LIN {X 0,Y 235.118,Z 411.198,A -85,B 0,C 180,E1 -19815.606,E2 -19815.606} C_VEL
LIN {X 0,Y 235.013,Z 411.211,A -85,B 0,C 180,E1 -19819.205,E2 -19819.205} C_VEL
LIN {X 0,Y 234.964,Z 411.217,A -85,B 0,C 180,E1 -19822.882,E2 -19822.882} C_VEL
LIN {X 0,Y 234.971,Z 411.217,A -85,B 0,C 180,E1 -19826.657,E2 -19826.657} C_VEL
LIN {X 0,Y 234.956,Z 411.22,A -85,B 0,C 180,E1 -19831.565,E2 -19831.565} C_VEL
LIN {X 0,Y 234.996,Z 411.371,A -85,B 0,C 180,E1 -19832.57,E2 -19832.57} C_VEL
LIN {X 0,Y 235.541,Z 414.614,A -85,B 0,C 180,E1 -19836.638,E2 -19836.638} C_VEL
LIN {X 0,Y 236.198,Z 418.359,A -85,B 0,C 180,E1 -19840.89,E2 -19840.89} C_VEL
LIN {X 0,Y 237.06,Z 422.615,A -85,B 0,C 180,E1 -19845.359,E2 -19845.359} C_VEL
LIN {X 0,Y 237.901,Z 427.546,A -85,B 0,C 180,E1 -19850.116,E2 -19850.116} C_VEL
LIN {X 0,Y 237.366,Z 428.622,A -85,B 0,C 180,E1 -19851.017,E2 -19851.017} C_VEL
LIN {X 0,Y 234.575,Z 430.575,A -85,B 0,C 180,E1 -19852.411,E2 -19852.411} C_VEL
LIN {X 0,Y 231.461,Z 432.564,A -85,B 0,C 180,E1 -19853.829,E2 -19853.829} C_VEL
LIN {X 0,Y 230.488,Z 433.723,A -85,B 0,C 180,E1 -19854.763,E2 -19854.763} C_VEL
LIN {X 0,Y 229.679,Z 436.812,A -85,B 0,C 180,E1 -19857.317,E2 -19857.317} C_VEL
LIN {X 0,Y 233.039,Z 450.186,A -85,B 0,C 180,E1 -19858.643,E2 -19858.643} C_VEL
LIN {X 0,Y 235.255,Z 462.15,A -85,B 0,C 180,E1 -19860.037,E2 -19860.037} C_VEL
LIN {X 0,Y 236.595,Z 473.99,A -85,B 0,C 180,E1 -19861.622,E2 -19861.622} C_VEL
LIN {X 0,Y 236.992,Z 485.015,A -85,B 0,C 180,E1 -19863.322,E2 -19863.322} C_VEL
LIN {X 0,Y 236.731,Z 495.453,A -85,B 0,C 180,E1 -19865.207,E2 -19865.207} C_VEL
LIN {X 0,Y 236.31,Z 498.762,A -85,B 0,C 180,E1 -19865.862,E2 -19865.862} C_VEL
LIN {X 0,Y 233.809,Z 508.392,A -85,B 0,C 180,E1 -19867.93,E2 -19867.93} C_VEL
LIN {X 0,Y 231.727,Z 516.41,A -85,B 0,C 180,E1 -19870.084,E2 -19870.084} C_VEL
LIN {X 0,Y 230.132,Z 522.879,A -85,B 0,C 180,E1 -19872.218,E2 -19872.218} C_VEL
LIN {X 0,Y 228.425,Z 529.354,A -85,B 0,C 180,E1 -19874.839,E2 -19874.839} C_VEL
LIN {X 0,Y 227.129,Z 534.507,A -85,B 0,C 180,E1 -19877.49,E2 -19877.49} C_VEL
LIN {X 0,Y 226.362,Z 538.526,A -85,B 0,C 180,E1 -19880.168,E2 -19880.168} C_VEL
LIN {X 0,Y 225.939,Z 541.504,A -85,B 0,C 180,E1 -19882.852,E2 -19882.852} C_VEL
LIN {X 0,Y 225.846,Z 542.993,A -85,B 0,C 180,E1 -19884.744,E2 -19884.744} C_VEL
LIN {X 0,Y 225.859,Z 543.948,A -85,B 0,C 180,E1 -19886.432,E2 -19886.432} C_VEL
LIN {X 0,Y 225.897,Z 544.572,A -85,B 0,C 180,E1 -19888.217,E2 -19888.217} C_VEL
LIN {X 0,Y 225.952,Z 544.793,A -85,B 0,C 180,E1 -19890,E2 -19890} C_VEL
LIN {X 0,Y 225.906,Z 544.564,A -85,B 0,C 180,E1 -19891.783,E2 -19891.783} C_VEL
LIN {X 0,Y 225.859,Z 543.936,A -85,B 0,C 180,E1 -19893.568,E2 -19893.568} C_VEL
LIN {X 0,Y 225.853,Z 542.911,A -85,B 0,C 180,E1 -19895.356,E2 -19895.356} C_VEL
LIN {X 0,Y 225.936,Z 541.479,A -85,B 0,C 180,E1 -19897.147,E2 -19897.147} C_VEL
LIN {X 0,Y 226.357,Z 538.489,A -85,B 0,C 180,E1 -19899.832,E2 -19899.832} C_VEL
LIN {X 0,Y 227.129,Z 534.455,A -85,B 0,C 180,E1 -19902.509,E2 -19902.509} C_VEL
LIN {X 0,Y 228.666,Z 528.278,A -85,B 0,C 180,E1 -19905.6,E2 -19905.6} C_VEL
LIN {X 0,Y 230.505,Z 521.548,A -85,B 0,C 180,E1 -19908.211,E2 -19908.211} C_VEL
LIN {X 0,Y 232.564,Z 513.252,A -85,B 0,C 180,E1 -19910.782,E2 -19910.782} C_VEL
LIN {X 0,Y 234.737,Z 504.655,A -85,B 0,C 180,E1 -19912.906,E2 -19912.906} C_VEL
LIN {X 0,Y 236.684,Z 496.44,A -85,B 0,C 180,E1 -19914.564,E2 -19914.564} C_VEL
LIN {X 0,Y 236.96,Z 486.42,A -85,B 0,C 180,E1 -19916.416,E2 -19916.416} C_VEL
LIN {X 0,Y 236.641,Z 475.292,A -85,B 0,C 180,E1 -19918.159,E2 -19918.159} C_VEL
LIN {X 0,Y 235.592,Z 464.68,A -85,B 0,C 180,E1 -19919.606,E2 -19919.606} C_VEL
LIN {X 0,Y 233.4,Z 451.947,A -85,B 0,C 180,E1 -19921.119,E2 -19921.119} C_VEL
LIN {X 0,Y 230.374,Z 439.737,A -85,B 0,C 180,E1 -19922.385,E2 -19922.385} C_VEL
LIN {X 0,Y 229.69,Z 436.608,A -85,B 0,C 180,E1 -19922.656,E2 -19922.656} C_VEL
LIN {X 0,Y 230.805,Z 432.292,A -85,B 0,C 180,E1 -19926.425,E2 -19926.425} C_VEL
LIN {X 0,Y 231.009,Z 429.893,A -85,B 0,C 180,E1 -19928.63,E2 -19928.63} C_VEL
LIN {X 0,Y 230.496,Z 426.268,A -85,B 0,C 180,E1 -19932.129,E2 -19932.129} C_VEL
LIN {X 0,Y 229.891,Z 423.154,A -85,B 0,C 180,E1 -19935.321,E2 -19935.321} C_VEL
LIN {X 0,Y 229.499,Z 420.96,A -85,B 0,C 180,E1 -19937.646,E2 -19937.646} C_VEL
LIN {X 0,Y 228.743,Z 417.112,A -85,B 0,C 180,E1 -19942.085,E2 -19942.085} C_VEL
LIN {X 0,Y 228.206,Z 413.712,A -85,B 0,C 180,E1 -19946.335,E2 -19946.335} C_VEL
LIN {X 0,Y 227.914,Z 412.092,A -85,B 0,C 180,E1 -19948.758,E2 -19948.758} C_VEL
LIN {X 0,Y 227.945,Z 412.092,A -85,B 0,C 180,E1 -19953.397,E2 -19953.397} C_VEL
LIN {X 0,Y 227.964,Z 412.09,A -85,B 0,C 180,E1 -19958.287,E2 -19958.287} C_VEL
LIN {X 0,Y 228.037,Z 412.08,A -85,B 0,C 180,E1 -19962.826,E2 -19962.826} C_VEL
LIN {X 0,Y 228.097,Z 412.073,A -85,B 0,C 180,E1 -19967.545,E2 -19967.545} C_VEL
LIN {X 0,Y 228.328,Z 412.044,A -85,B 0,C 180,E1 -19971.147,E2 -19971.147} C_VEL
LIN {X 0,Y 228.361,Z 412.041,A -85,B 0,C 180,E1 -19972.929,E2 -19972.929} C_VEL
LIN {X 0,Y 228.557,Z 412.016,A -85,B 0,C 180,E1 -19978.238,E2 -19978.238} C_VEL
LIN {X 0,Y 228.557,Z 412.013,A -85,B 0,C 180,E1 -19981.762,E2 -19981.762} C_VEL
LIN {X 0,Y 228.361,Z 412.036,A -85,B 0,C 180,E1 -19987.071,E2 -19987.071} C_VEL
LIN {X 0,Y 228.174,Z 412.063,A -85,B 0,C 180,E1 -19990.65,E2 -19990.65} C_VEL
LIN {X 0,Y 228.06,Z 412.076,A -85,B 0,C 180,E1 -19996.102,E2 -19996.102} C_VEL
LIN {X 0,Y 227.94,Z 412.091,A -85,B 0,C 180,E1 -19999.826,E2 -19999.826} C_VEL
LIN {X 0,Y 227.909,Z 412.096,A -85,B 0,C 180,E1 -20003.633,E2 -20003.633} C_VEL
LIN {X 0,Y 227.881,Z 412.098,A -85,B 0,C 180,E1 -20007.556,E2 -20007.556} C_VEL
LIN {X 0,Y 227.871,Z 412.099,A -85,B 0,C 180,E1 -20011.622,E2 -20011.622} C_VEL
LIN {X 0,Y 227.902,Z 412.094,A -85,B 0,C 180,E1 -20015.868,E2 -20015.868} C_VEL
LIN {X 0,Y 227.837,Z 412.102,A -85,B 0,C 180,E1 -20020.375,E2 -20020.375} C_VEL
LIN {X 0,Y 227.852,Z 412.102,A -85,B 0,C 180,E1 -20024.812,E2 -20024.812} C_VEL
LIN {X 0,Y 227.911,Z 412.097,A -85,B 0,C 180,E1 -20027.738,E2 -20027.738} C_VEL
LIN {X 0,Y 227.823,Z 412.11,A -85,B 0,C 180,E1 -20031.905,E2 -20031.905} C_VEL
LIN {X 0,Y 227.786,Z 412.217,A -85,B 0,C 180,E1 -20033.34,E2 -20033.34} C_VEL
LIN {X 0,Y 227.764,Z 414.508,A -85,B 0,C 180,E1 -20037.127,E2 -20037.127} C_VEL
LIN {X 0,Y 228.864,Z 417.579,A -85,B 0,C 180,E1 -20037.506,E2 -20037.506} C_VEL
LIN {X 0,Y 233.27,Z 427.972,A -85,B 0,C 180,E1 -20038.94,E2 -20038.94} C_VEL
LIN {X 0,Y 236.843,Z 438.708,A -85,B 0,C 180,E1 -20040.512,E2 -20040.512} C_VEL
LIN {X 0,Y 239.673,Z 450.577,A -85,B 0,C 180,E1 -20042.4,E2 -20042.4} C_VEL
LIN {X 0,Y 241.045,Z 460.006,A -85,B 0,C 180,E1 -20044.065,E2 -20044.065} C_VEL
LIN {X 0,Y 238.939,Z 470.189,A -85,B 0,C 180,E1 -20045.758,E2 -20045.758} C_VEL
LIN {X 0,Y 236.722,Z 479.756,A -85,B 0,C 180,E1 -20047.757,E2 -20047.757} C_VEL
LIN {X 0,Y 234.151,Z 489.351,A -85,B 0,C 180,E1 -20050.265,E2 -20050.265} C_VEL
LIN {X 0,Y 231.96,Z 496.993,A -85,B 0,C 180,E1 -20052.818,E2 -20052.818} C_VEL
LIN {X 0,Y 230.473,Z 502.204,A -85,B 0,C 180,E1 -20054.978,E2 -20054.978} C_VEL
LIN {X 0,Y 228.889,Z 507.261,A -85,B 0,C 180,E1 -20057.588,E2 -20057.588} C_VEL
LIN {X 0,Y 227.805,Z 511.175,A -85,B 0,C 180,E1 -20060.231,E2 -20060.231} C_VEL
LIN {X 0,Y 226.998,Z 514.065,A -85,B 0,C 180,E1 -20062.886,E2 -20062.886} C_VEL
LIN {X 0,Y 226.618,Z 515.446,A -85,B 0,C 180,E1 -20064.662,E2 -20064.662} C_VEL
LIN {X 0,Y 226.134,Z 517.035,A -85,B 0,C 180,E1 -20068.219,E2 -20068.219} C_VEL
LIN {X 0,Y 226.083,Z 517.262,A -85,B 0,C 180,E1 -20070,E2 -20070} C_VEL
LIN {X 0,Y 226.314,Z 516.485,A -85,B 0,C 180,E1 -20073.561,E2 -20073.561} C_VEL
LIN {X 0,Y 226.612,Z 515.522,A -85,B 0,C 180,E1 -20075.339,E2 -20075.339} C_VEL
LIN {X 0,Y 227.291,Z 512.996,A -85,B 0,C 180,E1 -20078.322,E2 -20078.322} C_VEL
LIN {X 0,Y 228.432,Z 508.871,A -85,B 0,C 180,E1 -20081.536,E2 -20081.536} C_VEL
LIN {X 0,Y 229.826,Z 504.262,A -85,B 0,C 180,E1 -20084.161,E2 -20084.161} C_VEL
LIN {X 0,Y 231.901,Z 497.31,A -85,B 0,C 180,E1 -20087.187,E2 -20087.187} C_VEL
LIN {X 0,Y 234.112,Z 489.764,A -85,B 0,C 180,E1 -20089.739,E2 -20089.739} C_VEL
LIN {X 0,Y 236.748,Z 480.254,A -85,B 0,C 180,E1 -20092.241,E2 -20092.241} C_VEL
LIN {X 0,Y 238.908,Z 470.452,A -85,B 0,C 180,E1 -20094.321,E2 -20094.321} C_VEL
LIN {X 0,Y 241.097,Z 459.787,A -85,B 0,C 180,E1 -20096.097,E2 -20096.097} C_VEL
LIN {X 0,Y 239.611,Z 450.011,A -85,B 0,C 180,E1 -20097.82,E2 -20097.82} C_VEL
LIN {X 0,Y 236.742,Z 438.204,A -85,B 0,C 180,E1 -20099.696,E2 -20099.696} C_VEL
LIN {X 0,Y 232.906,Z 426.871,A -85,B 0,C 180,E1 -20101.349,E2 -20101.349} C_VEL
LIN {X 0,Y 228.834,Z 417.379,A -85,B 0,C 180,E1 -20102.653,E2 -20102.653} C_VEL
LIN {X 0,Y 227.826,Z 414.457,A -85,B 0,C 180,E1 -20103.011,E2 -20103.011} C_VEL
LIN {X 0,Y 227.808,Z 412.296,A -85,B 0,C 180,E1 -20106.667,E2 -20106.667} C_VEL
LIN {X 0,Y 227.812,Z 412.109,A -85,B 0,C 180,E1 -20110.38,E2 -20110.38} C_VEL
LIN {X 0,Y 227.836,Z 412.102,A -85,B 0,C 180,E1 -20115.193,E2 -20115.193} C_VEL
LIN {X 0,Y 227.836,Z 412.105,A -85,B 0,C 180,E1 -20119.625,E2 -20119.625} C_VEL
LIN {X 0,Y 227.903,Z 412.093,A -85,B 0,C 180,E1 -20124.132,E2 -20124.132} C_VEL
LIN {X 0,Y 227.872,Z 412.102,A -85,B 0,C 180,E1 -20128.378,E2 -20128.378} C_VEL
LIN {X 0,Y 227.882,Z 412.099,A -85,B 0,C 180,E1 -20132.444,E2 -20132.444} C_VEL
LIN {X 0,Y 227.91,Z 412.096,A -85,B 0,C 180,E1 -20136.367,E2 -20136.367} C_VEL
LIN {X 0,Y 227.941,Z 412.091,A -85,B 0,C 180,E1 -20140.174,E2 -20140.174} C_VEL
LIN {X 0,Y 228.062,Z 412.076,A -85,B 0,C 180,E1 -20143.898,E2 -20143.898} C_VEL
LIN {X 0,Y 228.095,Z 412.072,A -85,B 0,C 180,E1 -20147.544,E2 -20147.544} C_VEL
LIN {X 0,Y 228.267,Z 412.051,A -85,B 0,C 180,E1 -20151.144,E2 -20151.144} C_VEL
LIN {X 0,Y 228.323,Z 412.043,A -85,B 0,C 180,E1 -20152.927,E2 -20152.927} C_VEL
LIN {X 0,Y 228.558,Z 412.016,A -85,B 0,C 180,E1 -20158.238,E2 -20158.238} C_VEL
LIN {X 0,Y 228.559,Z 412.018,A -85,B 0,C 180,E1 -20161.762,E2 -20161.762} C_VEL
LIN {X 0,Y 228.362,Z 412.039,A -85,B 0,C 180,E1 -20167.071,E2 -20167.071} C_VEL
LIN {X 0,Y 228.175,Z 412.063,A -85,B 0,C 180,E1 -20170.65,E2 -20170.65} C_VEL
LIN {X 0,Y 228.061,Z 412.074,A -85,B 0,C 180,E1 -20176.102,E2 -20176.102} C_VEL
LIN {X 0,Y 227.946,Z 412.09,A -85,B 0,C 180,E1 -20179.825,E2 -20179.825} C_VEL
LIN {X 0,Y 227.917,Z 412.095,A -85,B 0,C 180,E1 -20183.632,E2 -20183.632} C_VEL
LIN {X 0,Y 227.882,Z 412.101,A -85,B 0,C 180,E1 -20187.556,E2 -20187.556} C_VEL
LIN {X 0,Y 227.95,Z 412.221,A -85,B 0,C 180,E1 -20191.61,E2 -20191.61} C_VEL
LIN {X 0,Y 228.488,Z 415.401,A -85,B 0,C 180,E1 -20195.762,E2 -20195.762} C_VEL
LIN {X 0,Y 229.098,Z 419.034,A -85,B 0,C 180,E1 -20200.107,E2 -20200.107} C_VEL
LIN {X 0,Y 229.587,Z 421.382,A -85,B 0,C 180,E1 -20202.72,E2 -20202.72} C_VEL
LIN {X 0,Y 230.35,Z 425.541,A -85,B 0,C 180,E1 -20207.075,E2 -20207.075} C_VEL
LIN {X 0,Y 230.905,Z 428.788,A -85,B 0,C 180,E1 -20210.269,E2 -20210.269} C_VEL
LIN {X 0,Y 231.004,Z 431.191,A -85,B 0,C 180,E1 -20212.52,E2 -20212.52} C_VEL
LIN {X 0,Y 230.488,Z 433.723,A -85,B 0,C 180,E1 -20214.763,E2 -20214.763} C_VEL
LIN {X 0,Y 230.081,Z 435.409,A -85,B 0,C 180,E1 -20215.603,E2 -20215.603} C_VEL
LIN {X 0,Y 229.484,Z 438.755,A -85,B 0,C 180,E1 -20216.453,E2 -20216.453} C_VEL
LIN {X 0,Y 228.895,Z 442.891,A -85,B 0,C 180,E1 -20217.107,E2 -20217.107} C_VEL
LIN {X 0,Y 228.095,Z 452.58,A -85,B 0,C 180,E1 -20218.086,E2 -20218.086} C_VEL
LIN {X 0,Y 228.223,Z 458.488,A -85,B 0,C 180,E1 -20218.675,E2 -20218.675} C_VEL
LIN {X 0,Y 228.431,Z 460.389,A -85,B 0,C 180,E1 -20218.903,E2 -20218.903} C_VEL
LIN {X 0,Y 229.805,Z 472.029,A -85,B 0,C 180,E1 -20220.494,E2 -20220.494} C_VEL
LIN {X 0,Y 230.375,Z 482.933,A -85,B 0,C 180,E1 -20222.215,E2 -20222.215} C_VEL
LIN {X 0,Y 230.12,Z 493.812,A -85,B 0,C 180,E1 -20224.201,E2 -20224.201} C_VEL
LIN {X 0,Y 229.555,Z 499.407,A -85,B 0,C 180,E1 -20225.345,E2 -20225.345} C_VEL
LIN {X 0,Y 227.205,Z 507.96,A -85,B 0,C 180,E1 -20227.253,E2 -20227.253} C_VEL
LIN {X 0,Y 224.84,Z 516.64,A -85,B 0,C 180,E1 -20229.675,E2 -20229.675} C_VEL
LIN {X 0,Y 223.37,Z 522.447,A -85,B 0,C 180,E1 -20231.661,E2 -20231.661} C_VEL
LIN {X 0,Y 221.524,Z 528.92,A -85,B 0,C 180,E1 -20234.355,E2 -20234.355} C_VEL
LIN {X 0,Y 220.144,Z 534.072,A -85,B 0,C 180,E1 -20237.087,E2 -20237.087} C_VEL
LIN {X 0,Y 219.339,Z 538.092,A -85,B 0,C 180,E1 -20239.85,E2 -20239.85} C_VEL
LIN {X 0,Y 218.866,Z 541.07,A -85,B 0,C 180,E1 -20242.62,E2 -20242.62} C_VEL
LIN {X 0,Y 218.772,Z 542.697,A -85,B 0,C 180,E1 -20244.79,E2 -20244.79} C_VEL
LIN {X 0,Y 218.827,Z 544.141,A -85,B 0,C 180,E1 -20248.159,E2 -20248.159} C_VEL
LIN {X 0,Y 218.88,Z 544.362,A -85,B 0,C 180,E1 -20250,E2 -20250} C_VEL
LIN {X 0,Y 218.836,Z 544.133,A -85,B 0,C 180,E1 -20251.84,E2 -20251.84} C_VEL
LIN {X 0,Y 218.772,Z 542.68,A -85,B 0,C 180,E1 -20255.209,E2 -20255.209} C_VEL
LIN {X 0,Y 218.863,Z 541.044,A -85,B 0,C 180,E1 -20257.38,E2 -20257.38} C_VEL
LIN {X 0,Y 219.334,Z 538.054,A -85,B 0,C 180,E1 -20260.15,E2 -20260.15} C_VEL
LIN {X 0,Y 220.144,Z 534.018,A -85,B 0,C 180,E1 -20262.913,E2 -20262.913} C_VEL
LIN {X 0,Y 221.813,Z 527.842,A -85,B 0,C 180,E1 -20266.095,E2 -20266.095} C_VEL
LIN {X 0,Y 223.752,Z 521.113,A -85,B 0,C 180,E1 -20268.781,E2 -20268.781} C_VEL
LIN {X 0,Y 225.499,Z 514.264,A -85,B 0,C 180,E1 -20271.002,E2 -20271.002} C_VEL
LIN {X 0,Y 227.688,Z 506.029,A -85,B 0,C 180,E1 -20273.176,E2 -20273.176} C_VEL
LIN {X 0,Y 229.926,Z 497.077,A -85,B 0,C 180,E1 -20275.094,E2 -20275.094} C_VEL
LIN {X 0,Y 230.343,Z 485.964,A -85,B 0,C 180,E1 -20277.237,E2 -20277.237} C_VEL
LIN {X 0,Y 230.065,Z 475.029,A -85,B 0,C 180,E1 -20279.012,E2 -20279.012} C_VEL
LIN {X 0,Y 228.644,Z 462.174,A -85,B 0,C 180,E1 -20280.825,E2 -20280.825} C_VEL
LIN {X 0,Y 226.247,Z 448.991,A -85,B 0,C 180,E1 -20282.423,E2 -20282.423} C_VEL
LIN {X 0,Y 222.99,Z 436.927,A -85,B 0,C 180,E1 -20283.718,E2 -20283.718} C_VEL
LIN {X 0,Y 222.909,Z 436.099,A -85,B 0,C 180,E1 -20283.822,E2 -20283.822} C_VEL
LIN {X 0,Y 223.786,Z 432.99,A -85,B 0,C 180,E1 -20286.634,E2 -20286.634} C_VEL
LIN {X 0,Y 223.967,Z 430.652,A -85,B 0,C 180,E1 -20288.873,E2 -20288.873} C_VEL
LIN {X 0,Y 223.426,Z 427.086,A -85,B 0,C 180,E1 -20292.462,E2 -20292.462} C_VEL
LIN {X 0,Y 222.671,Z 423.281,A -85,B 0,C 180,E1 -20296.547,E2 -20296.547} C_VEL
LIN {X 0,Y 221.98,Z 419.658,A -85,B 0,C 180,E1 -20300.713,E2 -20300.713} C_VEL
LIN {X 0,Y 221.379,Z 416.125,A -85,B 0,C 180,E1 -20305.15,E2 -20305.15} C_VEL
LIN {X 0,Y 220.886,Z 412.969,A -85,B 0,C 180,E1 -20309.662,E2 -20309.662} C_VEL
LIN {X 0,Y 220.897,Z 412.969,A -85,B 0,C 180,E1 -20313.55,E2 -20313.55} C_VEL
LIN {X 0,Y 220.88,Z 412.971,A -85,B 0,C 180,E1 -20317.554,E2 -20317.554} C_VEL
LIN {X 0,Y 220.986,Z 412.959,A -85,B 0,C 180,E1 -20322.571,E2 -20322.571} C_VEL
LIN {X 0,Y 221.029,Z 412.954,A -85,B 0,C 180,E1 -20327.14,E2 -20327.14} C_VEL
LIN {X 0,Y 221.261,Z 412.925,A -85,B 0,C 180,E1 -20330.862,E2 -20330.862} C_VEL
LIN {X 0,Y 221.314,Z 412.92,A -85,B 0,C 180,E1 -20332.702,E2 -20332.702} C_VEL
LIN {X 0,Y 221.515,Z 412.894,A -85,B 0,C 180,E1 -20338.182,E2 -20338.182} C_VEL
LIN {X 0,Y 221.515,Z 412.89,A -85,B 0,C 180,E1 -20341.818,E2 -20341.818} C_VEL
LIN {X 0,Y 221.314,Z 412.914,A -85,B 0,C 180,E1 -20347.298,E2 -20347.298} C_VEL
LIN {X 0,Y 221.119,Z 412.941,A -85,B 0,C 180,E1 -20350.994,E2 -20350.994} C_VEL
LIN {X 0,Y 221.019,Z 412.954,A -85,B 0,C 180,E1 -20356.63,E2 -20356.63} C_VEL
LIN {X 0,Y 220.887,Z 412.97,A -85,B 0,C 180,E1 -20360.487,E2 -20360.487} C_VEL
LIN {X 0,Y 220.864,Z 412.972,A -85,B 0,C 180,E1 -20364.436,E2 -20364.436} C_VEL
LIN {X 0,Y 220.829,Z 412.977,A -85,B 0,C 180,E1 -20368.515,E2 -20368.515} C_VEL
LIN {X 0,Y 220.825,Z 412.971,A -85,B 0,C 180,E1 -20372.755,E2 -20372.755} C_VEL
LIN {X 0,Y 220.84,Z 412.972,A -85,B 0,C 180,E1 -20377.288,E2 -20377.288} C_VEL
LIN {X 0,Y 220.801,Z 412.981,A -85,B 0,C 180,E1 -20381.946,E2 -20381.946} C_VEL
LIN {X 0,Y 220.869,Z 412.973,A -85,B 0,C 180,E1 -20387.043,E2 -20387.043} C_VEL
LIN {X 0,Y 220.841,Z 412.979,A -85,B 0,C 180,E1 -20390.47,E2 -20390.47} C_VEL
LIN {X 0,Y 220.755,Z 413.148,A -85,B 0,C 180,E1 -20392.779,E2 -20392.779} C_VEL
LIN {X 0,Y 220.751,Z 414.965,A -85,B 0,C 180,E1 -20395.952,E2 -20395.952} C_VEL
LIN {X 0,Y 221.944,Z 418.146,A -85,B 0,C 180,E1 -20396.363,E2 -20396.363} C_VEL
LIN {X 0,Y 225.947,Z 427.166,A -85,B 0,C 180,E1 -20397.698,E2 -20397.698} C_VEL
LIN {X 0,Y 229.884,Z 438.441,A -85,B 0,C 180,E1 -20399.439,E2 -20399.439} C_VEL
LIN {X 0,Y 232.573,Z 449.122,A -85,B 0,C 180,E1 -20401.204,E2 -20401.204} C_VEL
LIN {X 0,Y 234.284,Z 458.794,A -85,B 0,C 180,E1 -20402.97,E2 -20402.97} C_VEL
LIN {X 0,Y 234.397,Z 461.779,A -85,B 0,C 180,E1 -20403.513,E2 -20403.513} C_VEL
LIN {X 0,Y 232.165,Z 471.986,A -85,B 0,C 180,E1 -20405.309,E2 -20405.309} C_VEL
LIN {X 0,Y 229.742,Z 481.956,A -85,B 0,C 180,E1 -20407.518,E2 -20407.518} C_VEL
LIN {X 0,Y 227.511,Z 489.784,A -85,B 0,C 180,E1 -20409.664,E2 -20409.664} C_VEL
LIN {X 0,Y 225.198,Z 497.427,A -85,B 0,C 180,E1 -20412.285,E2 -20412.285} C_VEL
LIN {X 0,Y 223.649,Z 502.636,A -85,B 0,C 180,E1 -20414.508,E2 -20414.508} C_VEL
LIN {X 0,Y 221.98,Z 507.693,A -85,B 0,C 180,E1 -20417.196,E2 -20417.196} C_VEL
LIN {X 0,Y 220.829,Z 511.607,A -85,B 0,C 180,E1 -20419.919,E2 -20419.919} C_VEL
LIN {X 0,Y 219.972,Z 514.497,A -85,B 0,C 180,E1 -20422.658,E2 -20422.658} C_VEL
LIN {X 0,Y 219.582,Z 515.877,A -85,B 0,C 180,E1 -20424.49,E2 -20424.49} C_VEL
LIN {X 0,Y 219.063,Z 517.466,A -85,B 0,C 180,E1 -20428.162,E2 -20428.162} C_VEL
LIN {X 0,Y 219.007,Z 517.693,A -85,B 0,C 180,E1 -20430,E2 -20430} C_VEL
LIN {X 0,Y 219.256,Z 516.915,A -85,B 0,C 180,E1 -20433.676,E2 -20433.676} C_VEL
LIN {X 0,Y 219.576,Z 515.952,A -85,B 0,C 180,E1 -20435.51,E2 -20435.51} C_VEL
LIN {X 0,Y 220.247,Z 513.581,A -85,B 0,C 180,E1 -20438.427,E2 -20438.427} C_VEL
LIN {X 0,Y 221.096,Z 510.574,A -85,B 0,C 180,E1 -20440.995,E2 -20440.995} C_VEL
LIN {X 0,Y 222.435,Z 506.345,A -85,B 0,C 180,E1 -20443.708,E2 -20443.708} C_VEL
LIN {X 0,Y 224.498,Z 499.935,A -85,B 0,C 180,E1 -20446.833,E2 -20446.833} C_VEL
LIN {X 0,Y 226.586,Z 492.887,A -85,B 0,C 180,E1 -20449.478,E2 -20449.478} C_VEL
LIN {X 0,Y 229.252,Z 484.09,A -85,B 0,C 180,E1 -20452.058,E2 -20452.058} C_VEL
LIN {X 0,Y 231.591,Z 474.865,A -85,B 0,C 180,E1 -20454.235,E2 -20454.235} C_VEL
LIN {X 0,Y 233.763,Z 465.065,A -85,B 0,C 180,E1 -20456.085,E2 -20456.085} C_VEL
LIN {X 0,Y 234.557,Z 461.213,A -85,B 0,C 180,E1 -20456.708,E2 -20456.708} C_VEL
LIN {X 0,Y 233.244,Z 452.129,A -85,B 0,C 180,E1 -20458.4,E2 -20458.4} C_VEL
LIN {X 0,Y 230.924,Z 441.904,A -85,B 0,C 180,E1 -20460.143,E2 -20460.143} C_VEL
LIN {X 0,Y 227.328,Z 430.637,A -85,B 0,C 180,E1 -20461.917,E2 -20461.917} C_VEL
LIN {X 0,Y 223.04,Z 420.246,A -85,B 0,C 180,E1 -20463.465,E2 -20463.465} C_VEL
LIN {X 0,Y 220.921,Z 415.609,A -85,B 0,C 180,E1 -20464.119,E2 -20464.119} C_VEL
LIN {X 0,Y 220.782,Z 414.945,A -85,B 0,C 180,E1 -20464.206,E2 -20464.206} C_VEL
LIN {X 0,Y 220.763,Z 413.208,A -85,B 0,C 180,E1 -20467.262,E2 -20467.262} C_VEL
LIN {X 0,Y 220.775,Z 412.985,A -85,B 0,C 180,E1 -20470.182,E2 -20470.182} C_VEL
LIN {X 0,Y 220.776,Z 412.985,A -85,B 0,C 180,E1 -20474.454,E2 -20474.454} C_VEL
LIN {X 0,Y 220.777,Z 412.982,A -85,B 0,C 180,E1 -20478.049,E2 -20478.049} C_VEL
LIN {X 0,Y 220.835,Z 412.977,A -85,B 0,C 180,E1 -20482.795,E2 -20482.795} C_VEL
LIN {X 0,Y 220.827,Z 412.977,A -85,B 0,C 180,E1 -20487.245,E2 -20487.245} C_VEL
LIN {X 0,Y 220.83,Z 412.977,A -85,B 0,C 180,E1 -20491.485,E2 -20491.485} C_VEL
LIN {X 0,Y 220.865,Z 412.971,A -85,B 0,C 180,E1 -20495.565,E2 -20495.565} C_VEL
LIN {X 0,Y 220.888,Z 412.97,A -85,B 0,C 180,E1 -20499.513,E2 -20499.513} C_VEL
LIN {X 0,Y 221.02,Z 412.953,A -85,B 0,C 180,E1 -20503.37,E2 -20503.37} C_VEL
LIN {X 0,Y 221.091,Z 412.943,A -85,B 0,C 180,E1 -20509.005,E2 -20509.005} C_VEL
LIN {X 0,Y 221.258,Z 412.923,A -85,B 0,C 180,E1 -20512.7,E2 -20512.7} C_VEL
LIN {X 0,Y 221.516,Z 412.893,A -85,B 0,C 180,E1 -20518.182,E2 -20518.182} C_VEL
LIN {X 0,Y 221.517,Z 412.896,A -85,B 0,C 180,E1 -20521.818,E2 -20521.818} C_VEL
LIN {X 0,Y 221.315,Z 412.918,A -85,B 0,C 180,E1 -20527.298,E2 -20527.298} C_VEL
LIN {X 0,Y 221.121,Z 412.943,A -85,B 0,C 180,E1 -20530.994,E2 -20530.994} C_VEL
LIN {X 0,Y 221.02,Z 412.949,A -85,B 0,C 180,E1 -20536.629,E2 -20536.629} C_VEL
LIN {X 0,Y 220.896,Z 412.966,A -85,B 0,C 180,E1 -20540.486,E2 -20540.486} C_VEL
LIN {X 0,Y 220.871,Z 412.973,A -85,B 0,C 180,E1 -20544.435,E2 -20544.435} C_VEL
LIN {X 0,Y 220.83,Z 412.978,A -85,B 0,C 180,E1 -20548.515,E2 -20548.515} C_VEL
LIN {X 0,Y 220.871,Z 413.111,A -85,B 0,C 180,E1 -20550.605,E2 -20550.605} C_VEL
LIN {X 0,Y 221.384,Z 416.173,A -85,B 0,C 180,E1 -20554.85,E2 -20554.85} C_VEL
LIN {X 0,Y 221.992,Z 419.716,A -85,B 0,C 180,E1 -20559.285,E2 -20559.285} C_VEL
LIN {X 0,Y 222.797,Z 423.781,A -85,B 0,C 180,E1 -20563.946,E2 -20563.946} C_VEL
LIN {X 0,Y 223.432,Z 427.163,A -85,B 0,C 180,E1 -20567.562,E2 -20567.562} C_VEL
LIN {X 0,Y 223.962,Z 430.709,A -85,B 0,C 180,E1 -20571.126,E2 -20571.126} C_VEL
LIN {X 0,Y 223.773,Z 433.089,A -85,B 0,C 180,E1 -20573.363,E2 -20573.363} C_VEL
LIN {X 0,Y 222.901,Z 436.199,A -85,B 0,C 180,E1 -20576.177,E2 -20576.177} C_VEL
LIN {X 0,Y 223.781,Z 439.653,A -85,B 0,C 180,E1 -20576.514,E2 -20576.514} C_VEL
LIN {X 0,Y 226.918,Z 452.315,A -85,B 0,C 180,E1 -20577.914,E2 -20577.914} C_VEL
LIN {X 0,Y 228.431,Z 460.389,A -85,B 0,C 180,E1 -20578.903,E2 -20578.903} C_VEL
LIN {X 0,Y 228.512,Z 465.858,A -85,B 0,C 180,E1 -20579.528,E2 -20579.528} C_VEL
LIN {X 0,Y 226.642,Z 474.956,A -85,B 0,C 180,E1 -20580.489,E2 -20580.489} C_VEL
LIN {X 0,Y 224.738,Z 481.88,A -85,B 0,C 180,E1 -20581.337,E2 -20581.337} C_VEL
LIN {X 0,Y 223.829,Z 486.851,A -85,B 0,C 180,E1 -20582.114,E2 -20582.114} C_VEL
LIN {X 0,Y 223.732,Z 488.423,A -85,B 0,C 180,E1 -20582.405,E2 -20582.405} C_VEL
LIN {X 0,Y 223.106,Z 498.977,A -85,B 0,C 180,E1 -20584.583,E2 -20584.583} C_VEL
LIN {X 0,Y 220.656,Z 507.529,A -85,B 0,C 180,E1 -20586.538,E2 -20586.538} C_VEL
LIN {X 0,Y 218.396,Z 515.437,A -85,B 0,C 180,E1 -20588.775,E2 -20588.775} C_VEL
LIN {X 0,Y 216.633,Z 522.016,A -85,B 0,C 180,E1 -20591.069,E2 -20591.069} C_VEL
LIN {X 0,Y 214.663,Z 528.487,A -85,B 0,C 180,E1 -20593.842,E2 -20593.842} C_VEL
LIN {X 0,Y 213.178,Z 533.638,A -85,B 0,C 180,E1 -20596.657,E2 -20596.657} C_VEL
LIN {X 0,Y 212.336,Z 537.66,A -85,B 0,C 180,E1 -20599.511,E2 -20599.511} C_VEL
LIN {X 0,Y 211.818,Z 540.638,A -85,B 0,C 180,E1 -20602.373,E2 -20602.373} C_VEL
LIN {X 0,Y 211.688,Z 542.421,A -85,B 0,C 180,E1 -20604.873,E2 -20604.873} C_VEL
LIN {X 0,Y 211.758,Z 543.71,A -85,B 0,C 180,E1 -20608.098,E2 -20608.098} C_VEL
LIN {X 0,Y 211.81,Z 543.931,A -85,B 0,C 180,E1 -20610,E2 -20610} C_VEL
LIN {X 0,Y 211.765,Z 543.702,A -85,B 0,C 180,E1 -20611.902,E2 -20611.902} C_VEL
LIN {X 0,Y 211.693,Z 542.392,A -85,B 0,C 180,E1 -20615.145,E2 -20615.145} C_VEL
LIN {X 0,Y 211.816,Z 540.611,A -85,B 0,C 180,E1 -20617.627,E2 -20617.627} C_VEL
LIN {X 0,Y 212.332,Z 537.619,A -85,B 0,C 180,E1 -20620.489,E2 -20620.489} C_VEL
LIN {X 0,Y 213.178,Z 533.581,A -85,B 0,C 180,E1 -20623.343,E2 -20623.343} C_VEL
LIN {X 0,Y 214.972,Z 527.406,A -85,B 0,C 180,E1 -20626.622,E2 -20626.622} C_VEL
LIN {X 0,Y 216.976,Z 520.772,A -85,B 0,C 180,E1 -20629.352,E2 -20629.352} C_VEL
LIN {X 0,Y 219.232,Z 512.321,A -85,B 0,C 180,E1 -20632.128,E2 -20632.128} C_VEL
LIN {X 0,Y 221.703,Z 503.783,A -85,B 0,C 180,E1 -20634.337,E2 -20634.337} C_VEL
LIN {X 0,Y 223.192,Z 497.714,A -85,B 0,C 180,E1 -20635.656,E2 -20635.656} C_VEL
LIN {X 0,Y 223.686,Z 488.169,A -85,B 0,C 180,E1 -20637.609,E2 -20637.609} C_VEL
LIN {X 0,Y 223.593,Z 476.331,A -85,B 0,C 180,E1 -20639.673,E2 -20639.673} C_VEL
LIN {X 0,Y 222.441,Z 464.568,A -85,B 0,C 180,E1 -20641.454,E2 -20641.454} C_VEL
LIN {X 0,Y 220.297,Z 451.775,A -85,B 0,C 180,E1 -20643.129,E2 -20643.129} C_VEL
LIN {X 0,Y 216.997,Z 438.977,A -85,B 0,C 180,E1 -20644.639,E2 -20644.639} C_VEL
LIN {X 0,Y 216.25,Z 435.611,A -85,B 0,C 180,E1 -20645.027,E2 -20645.027} C_VEL
LIN {X 0,Y 216.768,Z 433.688,A -85,B 0,C 180,E1 -20646.856,E2 -20646.856} C_VEL
LIN {X 0,Y 216.937,Z 431.556,A -85,B 0,C 180,E1 -20648.966,E2 -20648.966} C_VEL
LIN {X 0,Y 216.321,Z 427.694,A -85,B 0,C 180,E1 -20653.021,E2 -20653.021} C_VEL
LIN {X 0,Y 215.638,Z 424.314,A -85,B 0,C 180,E1 -20656.81,E2 -20656.81} C_VEL
LIN {X 0,Y 214.876,Z 420.214,A -85,B 0,C 180,E1 -20661.718,E2 -20661.718} C_VEL
LIN {X 0,Y 214.316,Z 416.901,A -85,B 0,C 180,E1 -20666.119,E2 -20666.119} C_VEL
LIN {X 0,Y 213.826,Z 413.85,A -85,B 0,C 180,E1 -20670.731,E2 -20670.731} C_VEL
LIN {X 0,Y 213.804,Z 413.855,A -85,B 0,C 180,E1 -20674.702,E2 -20674.702} C_VEL
LIN {X 0,Y 213.815,Z 413.851,A -85,B 0,C 180,E1 -20678.804,E2 -20678.804} C_VEL
LIN {X 0,Y 213.946,Z 413.835,A -85,B 0,C 180,E1 -20682.804,E2 -20682.804} C_VEL
LIN {X 0,Y 213.984,Z 413.832,A -85,B 0,C 180,E1 -20686.709,E2 -20686.709} C_VEL
LIN {X 0,Y 214.199,Z 413.807,A -85,B 0,C 180,E1 -20690.558,E2 -20690.558} C_VEL
LIN {X 0,Y 214.251,Z 413.799,A -85,B 0,C 180,E1 -20692.46,E2 -20692.46} C_VEL
LIN {X 0,Y 214.449,Z 413.774,A -85,B 0,C 180,E1 -20698.122,E2 -20698.122} C_VEL
LIN {X 0,Y 214.557,Z 413.759,A -85,B 0,C 180,E1 -20700,E2 -20700} C_VEL
LIN {X 0,Y 214.449,Z 413.771,A -85,B 0,C 180,E1 -20701.878,E2 -20701.878} C_VEL
LIN {X 0,Y 214.251,Z 413.794,A -85,B 0,C 180,E1 -20707.54,E2 -20707.54} C_VEL
LIN {X 0,Y 214.05,Z 413.821,A -85,B 0,C 180,E1 -20711.362,E2 -20711.362} C_VEL
LIN {X 0,Y 213.936,Z 413.835,A -85,B 0,C 180,E1 -20715.237,E2 -20715.237} C_VEL
LIN {X 0,Y 213.838,Z 413.846,A -85,B 0,C 180,E1 -20719.188,E2 -20719.188} C_VEL
LIN {X 0,Y 213.813,Z 413.851,A -85,B 0,C 180,E1 -20723.231,E2 -20723.231} C_VEL
LIN {X 0,Y 213.831,Z 413.847,A -85,B 0,C 180,E1 -20727.45,E2 -20727.45} C_VEL
LIN {X 0,Y 213.772,Z 413.854,A -85,B 0,C 180,E1 -20731.737,E2 -20731.737} C_VEL
LIN {X 0,Y 213.754,Z 413.854,A -85,B 0,C 180,E1 -20736.287,E2 -20736.287} C_VEL
LIN {X 0,Y 213.732,Z 413.86,A -85,B 0,C 180,E1 -20741.121,E2 -20741.121} C_VEL
LIN {X 0,Y 213.813,Z 413.852,A -85,B 0,C 180,E1 -20746.349,E2 -20746.349} C_VEL
LIN {X 0,Y 213.793,Z 413.855,A -85,B 0,C 180,E1 -20749.12,E2 -20749.12} C_VEL
LIN {X 0,Y 213.731,Z 414.046,A -85,B 0,C 180,E1 -20752.109,E2 -20752.109} C_VEL
LIN {X 0,Y 213.742,Z 415.431,A -85,B 0,C 180,E1 -20754.665,E2 -20754.665} C_VEL
LIN {X 0,Y 214.925,Z 418.568,A -85,B 0,C 180,E1 -20755.102,E2 -20755.102} C_VEL
LIN {X 0,Y 218.782,Z 426.802,A -85,B 0,C 180,E1 -20756.421,E2 -20756.421} C_VEL
LIN {X 0,Y 222.467,Z 436.724,A -85,B 0,C 180,E1 -20758.038,E2 -20758.038} C_VEL
LIN {X 0,Y 225.324,Z 446.854,A -85,B 0,C 180,E1 -20759.776,E2 -20759.776} C_VEL
LIN {X 0,Y 227.453,Z 458.027,A -85,B 0,C 180,E1 -20761.865,E2 -20761.865} C_VEL
LIN {X 0,Y 227.976,Z 462.222,A -85,B 0,C 180,E1 -20762.706,E2 -20762.706} C_VEL
LIN {X 0,Y 225.535,Z 473.359,A -85,B 0,C 180,E1 -20764.751,E2 -20764.751} C_VEL
LIN {X 0,Y 223.221,Z 482.39,A -85,B 0,C 180,E1 -20766.824,E2 -20766.824} C_VEL
LIN {X 0,Y 220.894,Z 490.218,A -85,B 0,C 180,E1 -20769.027,E2 -20769.027} C_VEL
LIN {X 0,Y 218.464,Z 497.86,A -85,B 0,C 180,E1 -20771.72,E2 -20771.72} C_VEL
LIN {X 0,Y 216.824,Z 503.07,A -85,B 0,C 180,E1 -20774.007,E2 -20774.007} C_VEL
LIN {X 0,Y 215.07,Z 508.126,A -85,B 0,C 180,E1 -20776.777,E2 -20776.777} C_VEL
LIN {X 0,Y 213.851,Z 512.04,A -85,B 0,C 180,E1 -20779.587,E2 -20779.587} C_VEL
LIN {X 0,Y 212.961,Z 514.928,A -85,B 0,C 180,E1 -20782.415,E2 -20782.415} C_VEL
LIN {X 0,Y 212.549,Z 516.307,A -85,B 0,C 180,E1 -20784.307,E2 -20784.307} C_VEL
LIN {X 0,Y 211.994,Z 517.897,A -85,B 0,C 180,E1 -20788.1,E2 -20788.1} C_VEL
LIN {X 0,Y 211.934,Z 518.124,A -85,B 0,C 180,E1 -20790,E2 -20790} C_VEL
LIN {X 0,Y 212.202,Z 517.346,A -85,B 0,C 180,E1 -20793.798,E2 -20793.798} C_VEL
LIN {X 0,Y 212.543,Z 516.382,A -85,B 0,C 180,E1 -20795.693,E2 -20795.693} C_VEL
LIN {X 0,Y 213.2,Z 514.174,A -85,B 0,C 180,E1 -20798.53,E2 -20798.53} C_VEL
LIN {X 0,Y 214.133,Z 511.006,A -85,B 0,C 180,E1 -20801.357,E2 -20801.357} C_VEL
LIN {X 0,Y 215.544,Z 506.776,A -85,B 0,C 180,E1 -20804.155,E2 -20804.155} C_VEL
LIN {X 0,Y 217.734,Z 500.364,A -85,B 0,C 180,E1 -20807.372,E2 -20807.372} C_VEL
LIN {X 0,Y 219.905,Z 493.318,A -85,B 0,C 180,E1 -20810.094,E2 -20810.094} C_VEL
LIN {X 0,Y 222.711,Z 484.518,A -85,B 0,C 180,E1 -20812.742,E2 -20812.742} C_VEL
LIN {X 0,Y 225.063,Z 475.652,A -85,B 0,C 180,E1 -20814.894,E2 -20814.894} C_VEL
LIN {X 0,Y 227.422,Z 465.491,A -85,B 0,C 180,E1 -20816.87,E2 -20816.87} C_VEL
LIN {X 0,Y 227.978,Z 462.925,A -85,B 0,C 180,E1 -20817.295,E2 -20817.295} C_VEL
LIN {X 0,Y 226.828,Z 453.99,A -85,B 0,C 180,E1 -20819.047,E2 -20819.047} C_VEL
LIN {X 0,Y 224.74,Z 444.312,A -85,B 0,C 180,E1 -20820.799,E2 -20820.799} C_VEL
LIN {X 0,Y 221.309,Z 433.217,A -85,B 0,C 180,E1 -20822.675,E2 -20822.675} C_VEL
LIN {X 0,Y 217.136,Z 422.819,A -85,B 0,C 180,E1 -20824.341,E2 -20824.341} C_VEL
LIN {X 0,Y 213.92,Z 416.177,A -85,B 0,C 180,E1 -20825.395,E2 -20825.395} C_VEL
LIN {X 0,Y 213.742,Z 415.425,A -85,B 0,C 180,E1 -20825.526,E2 -20825.526} C_VEL
LIN {X 0,Y 213.683,Z 413.869,A -85,B 0,C 180,E1 -20828.676,E2 -20828.676} C_VEL
LIN {X 0,Y 213.706,Z 413.864,A -85,B 0,C 180,E1 -20831.127,E2 -20831.127} C_VEL
LIN {X 0,Y 213.707,Z 413.864,A -85,B 0,C 180,E1 -20833.679,E2 -20833.679} C_VEL
LIN {X 0,Y 213.71,Z 413.865,A -85,B 0,C 180,E1 -20836.344,E2 -20836.344} C_VEL
LIN {X 0,Y 213.739,Z 413.856,A -85,B 0,C 180,E1 -20841.336,E2 -20841.336} C_VEL
LIN {X 0,Y 213.772,Z 413.855,A -85,B 0,C 180,E1 -20846.02,E2 -20846.02} C_VEL
LIN {X 0,Y 213.763,Z 413.858,A -85,B 0,C 180,E1 -20850.451,E2 -20850.451} C_VEL
LIN {X 0,Y 213.801,Z 413.85,A -85,B 0,C 180,E1 -20854.701,E2 -20854.701} C_VEL
LIN {X 0,Y 213.807,Z 413.852,A -85,B 0,C 180,E1 -20858.803,E2 -20858.803} C_VEL
LIN {X 0,Y 213.947,Z 413.833,A -85,B 0,C 180,E1 -20862.804,E2 -20862.804} C_VEL
LIN {X 0,Y 213.983,Z 413.828,A -85,B 0,C 180,E1 -20866.708,E2 -20866.708} C_VEL
LIN {X 0,Y 214.143,Z 413.811,A -85,B 0,C 180,E1 -20870.555,E2 -20870.555} C_VEL
LIN {X 0,Y 214.102,Z 413.817,A -85,B 0,C 180,E1 -20874.348,E2 -20874.348} C_VEL
LIN {X 0,Y 214.449,Z 413.774,A -85,B 0,C 180,E1 -20878.122,E2 -20878.122} C_VEL
LIN {X 0,Y 214.554,Z 413.763,A -85,B 0,C 180,E1 -20880,E2 -20880} C_VEL
LIN {X 0,Y 214.45,Z 413.776,A -85,B 0,C 180,E1 -20881.878,E2 -20881.878} C_VEL
LIN {X 0,Y 214.252,Z 413.8,A -85,B 0,C 180,E1 -20887.539,E2 -20887.539} C_VEL
LIN {X 0,Y 214.051,Z 413.822,A -85,B 0,C 180,E1 -20891.362,E2 -20891.362} C_VEL
LIN {X 0,Y 213.938,Z 413.837,A -85,B 0,C 180,E1 -20895.237,E2 -20895.237} C_VEL
LIN {X 0,Y 213.872,Z 413.844,A -85,B 0,C 180,E1 -20899.184,E2 -20899.184} C_VEL
LIN {X 0,Y 213.85,Z 413.848,A -85,B 0,C 180,E1 -20903.227,E2 -20903.227} C_VEL
LIN {X 0,Y 213.792,Z 413.855,A -85,B 0,C 180,E1 -20908.466,E2 -20908.466} C_VEL
LIN {X 0,Y 213.849,Z 413.986,A -85,B 0,C 180,E1 -20909.536,E2 -20909.536} C_VEL
LIN {X 0,Y 214.45,Z 417.764,A -85,B 0,C 180,E1 -20914.984,E2 -20914.984} C_VEL
LIN {X 0,Y 214.899,Z 420.412,A -85,B 0,C 180,E1 -20918.416,E2 -20918.416} C_VEL
LIN {X 0,Y 215.672,Z 424.363,A -85,B 0,C 180,E1 -20923.182,E2 -20923.182} C_VEL
LIN {X 0,Y 216.331,Z 427.774,A -85,B 0,C 180,E1 -20926.981,E2 -20926.981} C_VEL
LIN {X 0,Y 216.932,Z 431.624,A -85,B 0,C 180,E1 -20931.035,E2 -20931.035} C_VEL
LIN {X 0,Y 216.757,Z 433.777,A -85,B 0,C 180,E1 -20933.142,E2 -20933.142} C_VEL
LIN {X 0,Y 216.242,Z 435.721,A -85,B 0,C 180,E1 -20934.973,E2 -20934.973} C_VEL
LIN {X 0,Y 217.067,Z 439.164,A -85,B 0,C 180,E1 -20935.333,E2 -20935.333} C_VEL
LIN {X 0,Y 220.27,Z 451.634,A -85,B 0,C 180,E1 -20936.804,E2 -20936.804} C_VEL
LIN {X 0,Y 222.336,Z 463.457,A -85,B 0,C 180,E1 -20938.355,E2 -20938.355} C_VEL
LIN {X 0,Y 223.32,Z 473.075,A -85,B 0,C 180,E1 -20939.766,E2 -20939.766} C_VEL
LIN {X 0,Y 223.771,Z 482.219,A -85,B 0,C 180,E1 -20941.274,E2 -20941.274} C_VEL
LIN {X 0,Y 223.732,Z 488.423,A -85,B 0,C 180,E1 -20942.405,E2 -20942.405} C_VEL
LIN {X 0,Y 223.286,Z 491.639,A -85,B 0,C 180,E1 -20942.989,E2 -20942.989} C_VEL
LIN {X 0,Y 222.211,Z 494.822,A -85,B 0,C 180,E1 -20943.537,E2 -20943.537} C_VEL
LIN {X 0,Y 218.935,Z 500.854,A -85,B 0,C 180,E1 -20944.597,E2 -20944.597} C_VEL
LIN {X 0,Y 214.445,Z 507.984,A -85,B 0,C 180,E1 -20946.069,E2 -20946.069} C_VEL
LIN {X 0,Y 212.618,Z 511.998,A -85,B 0,C 180,E1 -20947.143,E2 -20947.143} C_VEL
LIN {X 0,Y 210.237,Z 520.486,A -85,B 0,C 180,E1 -20950.022,E2 -20950.022} C_VEL
LIN {X 0,Y 208.137,Z 527.051,A -85,B 0,C 180,E1 -20952.815,E2 -20952.815} C_VEL
LIN {X 0,Y 206.233,Z 533.204,A -85,B 0,C 180,E1 -20956.199,E2 -20956.199} C_VEL
LIN {X 0,Y 205.305,Z 537.225,A -85,B 0,C 180,E1 -20959.148,E2 -20959.148} C_VEL
LIN {X 0,Y 204.747,Z 540.204,A -85,B 0,C 180,E1 -20962.108,E2 -20962.108} C_VEL
LIN {X 0,Y 204.591,Z 542.167,A -85,B 0,C 180,E1 -20964.999,E2 -20964.999} C_VEL
LIN {X 0,Y 204.666,Z 543.278,A -85,B 0,C 180,E1 -20968.032,E2 -20968.032} C_VEL
LIN {X 0,Y 204.741,Z 543.501,A -85,B 0,C 180,E1 -20970,E2 -20970} C_VEL
LIN {X 0,Y 204.672,Z 543.27,A -85,B 0,C 180,E1 -20971.968,E2 -20971.968} C_VEL
LIN {X 0,Y 204.596,Z 542.138,A -85,B 0,C 180,E1 -20975.016,E2 -20975.016} C_VEL
LIN {X 0,Y 204.745,Z 540.176,A -85,B 0,C 180,E1 -20977.892,E2 -20977.892} C_VEL
LIN {X 0,Y 205.302,Z 537.183,A -85,B 0,C 180,E1 -20980.852,E2 -20980.852} C_VEL
LIN {X 0,Y 206.232,Z 533.145,A -85,B 0,C 180,E1 -20983.801,E2 -20983.801} C_VEL
LIN {X 0,Y 208.132,Z 526.969,A -85,B 0,C 180,E1 -20987.185,E2 -20987.185} C_VEL
LIN {X 0,Y 210.512,Z 519.303,A -85,B 0,C 180,E1 -20990.392,E2 -20990.392} C_VEL
LIN {X 0,Y 212.613,Z 511.883,A -85,B 0,C 180,E1 -20992.855,E2 -20992.855} C_VEL
LIN {X 0,Y 215.22,Z 503.345,A -85,B 0,C 180,E1 -20995.12,E2 -20995.12} C_VEL
LIN {X 0,Y 216.496,Z 498.352,A -85,B 0,C 180,E1 -20996.251,E2 -20996.251} C_VEL
LIN {X 0,Y 217.094,Z 488.442,A -85,B 0,C 180,E1 -20998.376,E2 -20998.376} C_VEL
LIN {X 0,Y 217.098,Z 477.483,A -85,B 0,C 180,E1 -21000.385,E2 -21000.385} C_VEL
LIN {X 0,Y 216.113,Z 465.754,A -85,B 0,C 180,E1 -21002.272,E2 -21002.272} C_VEL
LIN {X 0,Y 214.131,Z 453.283,A -85,B 0,C 180,E1 -21004.031,E2 -21004.031} C_VEL
LIN {X 0,Y 211.08,Z 441.146,A -85,B 0,C 180,E1 -21005.589,E2 -21005.589} C_VEL
LIN {X 0,Y 209.533,Z 435.195,A -85,B 0,C 180,E1 -21006.293,E2 -21006.293} C_VEL
LIN {X 0,Y 209.868,Z 433.195,A -85,B 0,C 180,E1 -21008.281,E2 -21008.281} C_VEL
LIN {X 0,Y 209.682,Z 430.817,A -85,B 0,C 180,E1 -21010.812,E2 -21010.812} C_VEL
LIN {X 0,Y 208.937,Z 427.042,A -85,B 0,C 180,E1 -21015.059,E2 -21015.059} C_VEL
LIN {X 0,Y 208.479,Z 424.679,A -85,B 0,C 180,E1 -21017.871,E2 -21017.871} C_VEL
LIN {X 0,Y 207.788,Z 421.017,A -85,B 0,C 180,E1 -21022.496,E2 -21022.496} C_VEL
LIN {X 0,Y 207.535,Z 419.286,A -85,B 0,C 180,E1 -21024.852,E2 -21024.852} C_VEL
LIN {X 0,Y 207.019,Z 416.194,A -85,B 0,C 180,E1 -21029.388,E2 -21029.388} C_VEL
LIN {X 0,Y 206.775,Z 414.728,A -85,B 0,C 180,E1 -21032.093,E2 -21032.093} C_VEL
LIN {X 0,Y 206.787,Z 414.728,A -85,B 0,C 180,E1 -21036.584,E2 -21036.584} C_VEL
LIN {X 0,Y 206.876,Z 414.717,A -85,B 0,C 180,E1 -21042.197,E2 -21042.197} C_VEL
LIN {X 0,Y 206.917,Z 414.714,A -85,B 0,C 180,E1 -21046.246,E2 -21046.246} C_VEL
LIN {X 0,Y 207.135,Z 414.686,A -85,B 0,C 180,E1 -21050.233,E2 -21050.233} C_VEL
LIN {X 0,Y 207.191,Z 414.677,A -85,B 0,C 180,E1 -21052.202,E2 -21052.202} C_VEL
LIN {X 0,Y 207.385,Z 414.654,A -85,B 0,C 180,E1 -21058.058,E2 -21058.058} C_VEL
LIN {X 0,Y 207.522,Z 414.635,A -85,B 0,C 180,E1 -21060,E2 -21060} C_VEL
LIN {X 0,Y 207.089,Z 414.689,A -85,B 0,C 180,E1 -21063.892,E2 -21063.892} C_VEL
LIN {X 0,Y 207.191,Z 414.674,A -85,B 0,C 180,E1 -21067.798,E2 -21067.798} C_VEL
LIN {X 0,Y 206.986,Z 414.703,A -85,B 0,C 180,E1 -21071.755,E2 -21071.755} C_VEL
LIN {X 0,Y 206.87,Z 414.715,A -85,B 0,C 180,E1 -21075.771,E2 -21075.771} C_VEL
LIN {X 0,Y 206.781,Z 414.727,A -85,B 0,C 180,E1 -21079.87,E2 -21079.87} C_VEL
LIN {X 0,Y 206.749,Z 414.731,A -85,B 0,C 180,E1 -21084.074,E2 -21084.074} C_VEL
LIN {X 0,Y 206.739,Z 414.733,A -85,B 0,C 180,E1 -21088.42,E2 -21088.42} C_VEL
LIN {X 0,Y 206.708,Z 414.729,A -85,B 0,C 180,E1 -21092.956,E2 -21092.956} C_VEL
LIN {X 0,Y 206.724,Z 414.735,A -85,B 0,C 180,E1 -21095.32,E2 -21095.32} C_VEL
LIN {X 0,Y 206.675,Z 414.737,A -85,B 0,C 180,E1 -21100.248,E2 -21100.248} C_VEL
LIN {X 0,Y 206.71,Z 414.738,A -85,B 0,C 180,E1 -21105.561,E2 -21105.561} C_VEL
LIN {X 0,Y 206.709,Z 414.737,A -85,B 0,C 180,E1 -21109.76,E2 -21109.76} C_VEL
LIN {X 0,Y 206.759,Z 415.419,A -85,B 0,C 180,E1 -21112.277,E2 -21112.277} C_VEL
LIN {X 0,Y 206.751,Z 415.945,A -85,B 0,C 180,E1 -21113.27,E2 -21113.27} C_VEL
LIN {X 0,Y 208.017,Z 419.212,A -85,B 0,C 180,E1 -21113.771,E2 -21113.771} C_VEL
LIN {X 0,Y 210.876,Z 424.914,A -85,B 0,C 180,E1 -21114.776,E2 -21114.776} C_VEL
LIN {X 0,Y 214.912,Z 434.803,A -85,B 0,C 180,E1 -21116.5,E2 -21116.5} C_VEL
LIN {X 0,Y 218.108,Z 445.17,A -85,B 0,C 180,E1 -21118.359,E2 -21118.359} C_VEL
LIN {X 0,Y 220.497,Z 456.381,A -85,B 0,C 180,E1 -21120.51,E2 -21120.51} C_VEL
LIN {X 0,Y 221.48,Z 463.936,A -85,B 0,C 180,E1 -21122.092,E2 -21122.092} C_VEL
LIN {X 0,Y 219.041,Z 474.229,A -85,B 0,C 180,E1 -21124.052,E2 -21124.052} C_VEL
LIN {X 0,Y 216.737,Z 482.824,A -85,B 0,C 180,E1 -21126.088,E2 -21126.088} C_VEL
LIN {X 0,Y 214.306,Z 490.651,A -85,B 0,C 180,E1 -21128.35,E2 -21128.35} C_VEL
LIN {X 0,Y 211.758,Z 498.293,A -85,B 0,C 180,E1 -21131.12,E2 -21131.12} C_VEL
LIN {X 0,Y 210.009,Z 503.504,A -85,B 0,C 180,E1 -21133.474,E2 -21133.474} C_VEL
LIN {X 0,Y 208.182,Z 508.559,A -85,B 0,C 180,E1 -21136.331,E2 -21136.331} C_VEL
LIN {X 0,Y 206.88,Z 512.473,A -85,B 0,C 180,E1 -21139.232,E2 -21139.232} C_VEL
LIN {X 0,Y 205.931,Z 515.361,A -85,B 0,C 180,E1 -21142.154,E2 -21142.154} C_VEL
LIN {X 0,Y 205.52,Z 516.738,A -85,B 0,C 180,E1 -21144.112,E2 -21144.112} C_VEL
LIN {X 0,Y 204.928,Z 518.328,A -85,B 0,C 180,E1 -21148.035,E2 -21148.035} C_VEL
LIN {X 0,Y 204.862,Z 518.555,A -85,B 0,C 180,E1 -21150,E2 -21150} C_VEL
LIN {X 0,Y 205.15,Z 517.776,A -85,B 0,C 180,E1 -21153.929,E2 -21153.929} C_VEL
LIN {X 0,Y 205.513,Z 516.812,A -85,B 0,C 180,E1 -21155.889,E2 -21155.889} C_VEL
LIN {X 0,Y 206.132,Z 514.802,A -85,B 0,C 180,E1 -21158.602,E2 -21158.602} C_VEL
LIN {X 0,Y 207.196,Z 511.436,A -85,B 0,C 180,E1 -21161.743,E2 -21161.743} C_VEL
LIN {X 0,Y 208.679,Z 507.206,A -85,B 0,C 180,E1 -21164.631,E2 -21164.631} C_VEL
LIN {X 0,Y 210.968,Z 500.794,A -85,B 0,C 180,E1 -21167.948,E2 -21167.948} C_VEL
LIN {X 0,Y 213.269,Z 493.746,A -85,B 0,C 180,E1 -21170.748,E2 -21170.748} C_VEL
LIN {X 0,Y 216.205,Z 484.946,A -85,B 0,C 180,E1 -21173.466,E2 -21173.466} C_VEL
LIN {X 0,Y 218.85,Z 475.335,A -85,B 0,C 180,E1 -21175.845,E2 -21175.845} C_VEL
LIN {X 0,Y 221.135,Z 465.918,A -85,B 0,C 180,E1 -21177.698,E2 -21177.698} C_VEL
LIN {X 0,Y 221.46,Z 463.369,A -85,B 0,C 180,E1 -21178.168,E2 -21178.168} C_VEL
LIN {X 0,Y 219.911,Z 452.678,A -85,B 0,C 180,E1 -21180.358,E2 -21180.358} C_VEL
LIN {X 0,Y 217.463,Z 442.494,A -85,B 0,C 180,E1 -21182.272,E2 -21182.272} C_VEL
LIN {X 0,Y 213.696,Z 431.316,A -85,B 0,C 180,E1 -21184.25,E2 -21184.25} C_VEL
LIN {X 0,Y 209.685,Z 422.407,A -85,B 0,C 180,E1 -21185.821,E2 -21185.821} C_VEL
LIN {X 0,Y 207.776,Z 418.772,A -85,B 0,C 180,E1 -21186.465,E2 -21186.465} C_VEL
LIN {X 0,Y 206.73,Z 415.946,A -85,B 0,C 180,E1 -21186.888,E2 -21186.888} C_VEL
LIN {X 0,Y 206.7,Z 415.089,A -85,B 0,C 180,E1 -21188.554,E2 -21188.554} C_VEL
LIN {X 0,Y 206.638,Z 414.745,A -85,B 0,C 180,E1 -21191.561,E2 -21191.561} C_VEL
LIN {X 0,Y 206.637,Z 414.743,A -85,B 0,C 180,E1 -21195.582,E2 -21195.582} C_VEL
LIN {X 0,Y 206.669,Z 414.742,A -85,B 0,C 180,E1 -21199.75,E2 -21199.75} C_VEL
LIN {X 0,Y 206.734,Z 414.728,A -85,B 0,C 180,E1 -21204.695,E2 -21204.695} C_VEL
LIN {X 0,Y 206.71,Z 414.736,A -85,B 0,C 180,E1 -21209.337,E2 -21209.337} C_VEL
LIN {X 0,Y 206.734,Z 414.734,A -85,B 0,C 180,E1 -21213.772,E2 -21213.772} C_VEL
LIN {X 0,Y 206.743,Z 414.731,A -85,B 0,C 180,E1 -21218.041,E2 -21218.041} C_VEL
LIN {X 0,Y 206.877,Z 414.716,A -85,B 0,C 180,E1 -21222.197,E2 -21222.197} C_VEL
LIN {X 0,Y 206.917,Z 414.709,A -85,B 0,C 180,E1 -21226.246,E2 -21226.246} C_VEL
LIN {X 0,Y 207.103,Z 414.689,A -85,B 0,C 180,E1 -21230.231,E2 -21230.231} C_VEL
LIN {X 0,Y 207.063,Z 414.694,A -85,B 0,C 180,E1 -21234.156,E2 -21234.156} C_VEL
LIN {X 0,Y 207.385,Z 414.654,A -85,B 0,C 180,E1 -21238.058,E2 -21238.058} C_VEL
LIN {X 0,Y 207.519,Z 414.639,A -85,B 0,C 180,E1 -21240,E2 -21240} C_VEL
LIN {X 0,Y 207.387,Z 414.657,A -85,B 0,C 180,E1 -21241.942,E2 -21241.942} C_VEL
LIN {X 0,Y 207.193,Z 414.68,A -85,B 0,C 180,E1 -21247.798,E2 -21247.798} C_VEL
LIN {X 0,Y 206.987,Z 414.702,A -85,B 0,C 180,E1 -21251.755,E2 -21251.755} C_VEL
LIN {X 0,Y 206.872,Z 414.715,A -85,B 0,C 180,E1 -21255.77,E2 -21255.77} C_VEL
LIN {X 0,Y 206.803,Z 414.724,A -85,B 0,C 180,E1 -21259.867,E2 -21259.867} C_VEL
LIN {X 0,Y 206.767,Z 414.73,A -85,B 0,C 180,E1 -21264.072,E2 -21264.072} C_VEL
LIN {X 0,Y 206.788,Z 414.876,A -85,B 0,C 180,E1 -21268.412,E2 -21268.412} C_VEL
LIN {X 0,Y 207.226,Z 417.758,A -85,B 0,C 180,E1 -21272.863,E2 -21272.863} C_VEL
LIN {X 0,Y 207.572,Z 419.719,A -85,B 0,C 180,E1 -21275.649,E2 -21275.649} C_VEL
LIN {X 0,Y 208.126,Z 422.961,A -85,B 0,C 180,E1 -21279.911,E2 -21279.911} C_VEL
LIN {X 0,Y 209.001,Z 427.089,A -85,B 0,C 180,E1 -21284.923,E2 -21284.923} C_VEL
LIN {X 0,Y 209.668,Z 430.892,A -85,B 0,C 180,E1 -21289.185,E2 -21289.185} C_VEL
LIN {X 0,Y 209.862,Z 433.282,A -85,B 0,C 180,E1 -21291.717,E2 -21291.717} C_VEL
LIN {X 0,Y 209.522,Z 435.263,A -85,B 0,C 180,E1 -21293.692,E2 -21293.692} C_VEL
LIN {X 0,Y 210.414,Z 438.692,A -85,B 0,C 180,E1 -21294.071,E2 -21294.071} C_VEL
LIN {X 0,Y 213.768,Z 451.56,A -85,B 0,C 180,E1 -21295.693,E2 -21295.693} C_VEL
LIN {X 0,Y 216.008,Z 464.423,A -85,B 0,C 180,E1 -21297.486,E2 -21297.486} C_VEL
LIN {X 0,Y 217.011,Z 476.137,A -85,B 0,C 180,E1 -21299.331,E2 -21299.331} C_VEL
LIN {X 0,Y 217.212,Z 485.283,A -85,B 0,C 180,E1 -21300.965,E2 -21300.965} C_VEL
LIN {X 0,Y 216.777,Z 495.265,A -85,B 0,C 180,E1 -21303.006,E2 -21303.006} C_VEL
LIN {X 0,Y 216.385,Z 499.588,A -85,B 0,C 180,E1 -21303.993,E2 -21303.993} C_VEL
LIN {X 0,Y 213.601,Z 508.777,A -85,B 0,C 180,E1 -21306.23,E2 -21306.23} C_VEL
LIN {X 0,Y 212.618,Z 511.998,A -85,B 0,C 180,E1 -21307.143,E2 -21307.143} C_VEL
LIN {X 0,Y 210.847,Z 515.807,A -85,B 0,C 180,E1 -21308.268,E2 -21308.268} C_VEL
LIN {X 0,Y 206.368,Z 521.472,A -85,B 0,C 180,E1 -21310.136,E2 -21310.136} C_VEL
LIN {X 0,Y 201.992,Z 526.533,A -85,B 0,C 180,E1 -21312.204,E2 -21312.204} C_VEL
LIN {X 0,Y 200.419,Z 529.302,A -85,B 0,C 180,E1 -21313.62,E2 -21313.62} C_VEL
LIN {X 0,Y 198.919,Z 534.222,A -85,B 0,C 180,E1 -21316.723,E2 -21316.723} C_VEL
LIN {X 0,Y 198.058,Z 537.88,A -85,B 0,C 180,E1 -21319.78,E2 -21319.78} C_VEL
LIN {X 0,Y 197.694,Z 539.771,A -85,B 0,C 180,E1 -21321.825,E2 -21321.825} C_VEL
LIN {X 0,Y 197.498,Z 541.894,A -85,B 0,C 180,E1 -21325.127,E2 -21325.127} C_VEL
LIN {X 0,Y 197.576,Z 542.847,A -85,B 0,C 180,E1 -21327.961,E2 -21327.961} C_VEL
LIN {X 0,Y 197.674,Z 543.07,A -85,B 0,C 180,E1 -21330,E2 -21330} C_VEL
LIN {X 0,Y 197.582,Z 542.838,A -85,B 0,C 180,E1 -21332.038,E2 -21332.038} C_VEL
LIN {X 0,Y 197.498,Z 541.877,A -85,B 0,C 180,E1 -21334.873,E2 -21334.873} C_VEL
LIN {X 0,Y 197.692,Z 539.741,A -85,B 0,C 180,E1 -21338.175,E2 -21338.175} C_VEL
LIN {X 0,Y 198.281,Z 536.746,A -85,B 0,C 180,E1 -21341.241,E2 -21341.241} C_VEL
LIN {X 0,Y 199.299,Z 532.708,A -85,B 0,C 180,E1 -21344.291,E2 -21344.291} C_VEL
LIN {X 0,Y 201.303,Z 526.532,A -85,B 0,C 180,E1 -21347.787,E2 -21347.787} C_VEL
LIN {X 0,Y 203.574,Z 519.669,A -85,B 0,C 180,E1 -21350.779,E2 -21350.779} C_VEL
LIN {X 0,Y 206.052,Z 511.445,A -85,B 0,C 180,E1 -21353.626,E2 -21353.626} C_VEL
LIN {X 0,Y 208.799,Z 502.909,A -85,B 0,C 180,E1 -21355.949,E2 -21355.949} C_VEL
LIN {X 0,Y 209.921,Z 497.901,A -85,B 0,C 180,E1 -21357.139,E2 -21357.139} C_VEL
LIN {X 0,Y 210.557,Z 487.994,A -85,B 0,C 180,E1 -21359.339,E2 -21359.339} C_VEL
LIN {X 0,Y 210.538,Z 477.007,A -85,B 0,C 180,E1 -21361.438,E2 -21361.438} C_VEL
LIN {X 0,Y 209.636,Z 465.522,A -85,B 0,C 180,E1 -21363.362,E2 -21363.362} C_VEL
LIN {X 0,Y 207.81,Z 453.967,A -85,B 0,C 180,E1 -21365.095,E2 -21365.095} C_VEL
LIN {X 0,Y 204.74,Z 441.369,A -85,B 0,C 180,E1 -21366.821,E2 -21366.821} C_VEL
LIN {X 0,Y 202.816,Z 435.154,A -85,B 0,C 180,E1 -21367.623,E2 -21367.623} C_VEL
LIN {X 0,Y 202.748,Z 434.678,A -85,B 0,C 180,E1 -21367.712,E2 -21367.712} C_VEL
LIN {X 0,Y 202.58,Z 431.489,A -85,B 0,C 180,E1 -21371.236,E2 -21371.236} C_VEL
LIN {X 0,Y 201.805,Z 427.588,A -85,B 0,C 180,E1 -21375.852,E2 -21375.852} C_VEL
LIN {X 0,Y 201.048,Z 423.522,A -85,B 0,C 180,E1 -21381.007,E2 -21381.007} C_VEL
LIN {X 0,Y 200.427,Z 420.061,A -85,B 0,C 180,E1 -21385.872,E2 -21385.872} C_VEL
LIN {X 0,Y 199.937,Z 417.062,A -85,B 0,C 180,E1 -21390.52,E2 -21390.52} C_VEL
LIN {X 0,Y 199.685,Z 415.613,A -85,B 0,C 180,E1 -21393.337,E2 -21393.337} C_VEL
LIN {X 0,Y 199.74,Z 415.604,A -85,B 0,C 180,E1 -21397.229,E2 -21397.229} C_VEL
LIN {X 0,Y 199.798,Z 415.598,A -85,B 0,C 180,E1 -21401.757,E2 -21401.757} C_VEL
LIN {X 0,Y 199.851,Z 415.592,A -85,B 0,C 180,E1 -21405.749,E2 -21405.749} C_VEL
LIN {X 0,Y 200.078,Z 415.563,A -85,B 0,C 180,E1 -21409.885,E2 -21409.885} C_VEL
LIN {X 0,Y 200.135,Z 415.556,A -85,B 0,C 180,E1 -21411.925,E2 -21411.925} C_VEL
LIN {X 0,Y 200.325,Z 415.533,A -85,B 0,C 180,E1 -21417.99,E2 -21417.99} C_VEL
LIN {X 0,Y 200.486,Z 415.511,A -85,B 0,C 180,E1 -21420,E2 -21420} C_VEL
LIN {X 0,Y 200.035,Z 415.567,A -85,B 0,C 180,E1 -21424.029,E2 -21424.029} C_VEL
LIN {X 0,Y 200.135,Z 415.555,A -85,B 0,C 180,E1 -21428.075,E2 -21428.075} C_VEL
LIN {X 0,Y 199.917,Z 415.582,A -85,B 0,C 180,E1 -21432.177,E2 -21432.177} C_VEL
LIN {X 0,Y 199.807,Z 415.595,A -85,B 0,C 180,E1 -21436.343,E2 -21436.343} C_VEL
LIN {X 0,Y 199.693,Z 415.61,A -85,B 0,C 180,E1 -21440.606,E2 -21440.606} C_VEL
LIN {X 0,Y 199.667,Z 415.612,A -85,B 0,C 180,E1 -21444.985,E2 -21444.985} C_VEL
LIN {X 0,Y 199.666,Z 415.613,A -85,B 0,C 180,E1 -21449.524,E2 -21449.524} C_VEL
LIN {X 0,Y 199.66,Z 415.607,A -85,B 0,C 180,E1 -21452.35,E2 -21452.35} C_VEL
LIN {X 0,Y 199.621,Z 415.613,A -85,B 0,C 180,E1 -21456.764,E2 -21456.764} C_VEL
LIN {X 0,Y 199.642,Z 415.616,A -85,B 0,C 180,E1 -21459.321,E2 -21459.321} C_VEL
LIN {X 0,Y 199.633,Z 415.618,A -85,B 0,C 180,E1 -21464.757,E2 -21464.757} C_VEL
LIN {X 0,Y 199.666,Z 415.615,A -85,B 0,C 180,E1 -21468.027,E2 -21468.027} C_VEL
LIN {X 0,Y 199.746,Z 416.261,A -85,B 0,C 180,E1 -21471.393,E2 -21471.393} C_VEL
LIN {X 0,Y 199.783,Z 416.593,A -85,B 0,C 180,E1 -21471.794,E2 -21471.794} C_VEL
LIN {X 0,Y 201.019,Z 419.665,A -85,B 0,C 180,E1 -21472.288,E2 -21472.288} C_VEL
LIN {X 0,Y 202.234,Z 421.853,A -85,B 0,C 180,E1 -21472.713,E2 -21472.713} C_VEL
LIN {X 0,Y 206.789,Z 431.65,A -85,B 0,C 180,E1 -21474.578,E2 -21474.578} C_VEL
LIN {X 0,Y 210.51,Z 442.24,A -85,B 0,C 180,E1 -21476.579,E2 -21476.579} C_VEL
LIN {X 0,Y 213.086,Z 452.41,A -85,B 0,C 180,E1 -21478.585,E2 -21478.585} C_VEL
LIN {X 0,Y 214.625,Z 461.843,A -85,B 0,C 180,E1 -21480.582,E2 -21480.582} C_VEL
LIN {X 0,Y 214.97,Z 465.652,A -85,B 0,C 180,E1 -21481.436,E2 -21481.436} C_VEL
LIN {X 0,Y 212.29,Z 476.242,A -85,B 0,C 180,E1 -21483.567,E2 -21483.567} C_VEL
LIN {X 0,Y 209.773,Z 484.938,A -85,B 0,C 180,E1 -21485.769,E2 -21485.769} C_VEL
LIN {X 0,Y 206.712,Z 493.81,A -85,B 0,C 180,E1 -21488.562,E2 -21488.562} C_VEL
LIN {X 0,Y 204.331,Z 500.931,A -85,B 0,C 180,E1 -21491.449,E2 -21491.449} C_VEL
LIN {X 0,Y 202.516,Z 505.735,A -85,B 0,C 180,E1 -21493.881,E2 -21493.881} C_VEL
LIN {X 0,Y 200.787,Z 510.397,A -85,B 0,C 180,E1 -21496.849,E2 -21496.849} C_VEL
LIN {X 0,Y 199.52,Z 513.958,A -85,B 0,C 180,E1 -21499.856,E2 -21499.856} C_VEL
LIN {X 0,Y 198.91,Z 515.793,A -85,B 0,C 180,E1 -21501.875,E2 -21501.875} C_VEL
LIN {X 0,Y 198.469,Z 517.17,A -85,B 0,C 180,E1 -21503.902,E2 -21503.902} C_VEL
LIN {X 0,Y 197.863,Z 518.759,A -85,B 0,C 180,E1 -21507.965,E2 -21507.965} C_VEL
LIN {X 0,Y 197.792,Z 518.985,A -85,B 0,C 180,E1 -21510,E2 -21510} C_VEL
LIN {X 0,Y 198.101,Z 518.206,A -85,B 0,C 180,E1 -21514.069,E2 -21514.069} C_VEL
LIN {X 0,Y 198.463,Z 517.243,A -85,B 0,C 180,E1 -21516.099,E2 -21516.099} C_VEL
LIN {X 0,Y 199.03,Z 515.489,A -85,B 0,C 180,E1 -21518.614,E2 -21518.614} C_VEL
LIN {X 0,Y 200.26,Z 511.866,A -85,B 0,C 180,E1 -21522.156,E2 -21522.156} C_VEL
LIN {X 0,Y 201.837,Z 507.636,A -85,B 0,C 180,E1 -21525.139,E2 -21525.139} C_VEL
LIN {X 0,Y 204.233,Z 501.224,A -85,B 0,C 180,E1 -21528.561,E2 -21528.561} C_VEL
LIN {X 0,Y 206.67,Z 494.175,A -85,B 0,C 180,E1 -21531.443,E2 -21531.443} C_VEL
LIN {X 0,Y 209.736,Z 485.374,A -85,B 0,C 180,E1 -21534.236,E2 -21534.236} C_VEL
LIN {X 0,Y 212.382,Z 476.181,A -85,B 0,C 180,E1 -21536.582,E2 -21536.582} C_VEL
LIN {X 0,Y 214.898,Z 466.344,A -85,B 0,C 180,E1 -21538.574,E2 -21538.574} C_VEL
LIN {X 0,Y 214.631,Z 461.452,A -85,B 0,C 180,E1 -21539.639,E2 -21539.639} C_VEL
LIN {X 0,Y 213.172,Z 452.428,A -85,B 0,C 180,E1 -21541.546,E2 -21541.546} C_VEL
LIN {X 0,Y 210.27,Z 441.193,A -85,B 0,C 180,E1 -21543.756,E2 -21543.756} C_VEL
LIN {X 0,Y 206.354,Z 430.436,A -85,B 0,C 180,E1 -21545.79,E2 -21545.79} C_VEL
LIN {X 0,Y 201.463,Z 420.308,A -85,B 0,C 180,E1 -21547.729,E2 -21547.729} C_VEL
LIN {X 0,Y 199.941,Z 417.358,A -85,B 0,C 180,E1 -21548.284,E2 -21548.284} C_VEL
LIN {X 0,Y 199.747,Z 416.44,A -85,B 0,C 180,E1 -21548.435,E2 -21548.435} C_VEL
LIN {X 0,Y 199.663,Z 416.019,A -85,B 0,C 180,E1 -21549.316,E2 -21549.316} C_VEL
LIN {X 0,Y 199.573,Z 415.627,A -85,B 0,C 180,E1 -21552.309,E2 -21552.309} C_VEL
LIN {X 0,Y 199.583,Z 415.621,A -85,B 0,C 180,E1 -21555.229,E2 -21555.229} C_VEL
LIN {X 0,Y 199.642,Z 415.612,A -85,B 0,C 180,E1 -21560.679,E2 -21560.679} C_VEL
LIN {X 0,Y 199.636,Z 415.614,A -85,B 0,C 180,E1 -21565.718,E2 -21565.718} C_VEL
LIN {X 0,Y 199.699,Z 415.609,A -85,B 0,C 180,E1 -21568.137,E2 -21568.137} C_VEL
LIN {X 0,Y 199.688,Z 415.61,A -85,B 0,C 180,E1 -21572.772,E2 -21572.772} C_VEL
LIN {X 0,Y 199.718,Z 415.606,A -85,B 0,C 180,E1 -21577.226,E2 -21577.226} C_VEL
LIN {X 0,Y 199.8,Z 415.597,A -85,B 0,C 180,E1 -21581.758,E2 -21581.758} C_VEL
LIN {X 0,Y 199.851,Z 415.59,A -85,B 0,C 180,E1 -21585.749,E2 -21585.749} C_VEL
LIN {X 0,Y 200.026,Z 415.568,A -85,B 0,C 180,E1 -21589.882,E2 -21589.882} C_VEL
LIN {X 0,Y 200.024,Z 415.572,A -85,B 0,C 180,E1 -21593.949,E2 -21593.949} C_VEL
LIN {X 0,Y 200.325,Z 415.533,A -85,B 0,C 180,E1 -21597.989,E2 -21597.989} C_VEL
LIN {X 0,Y 200.483,Z 415.516,A -85,B 0,C 180,E1 -21600,E2 -21600} C_VEL
LIN {X 0,Y 200.037,Z 415.57,A -85,B 0,C 180,E1 -21604.029,E2 -21604.029} C_VEL
LIN {X 0,Y 200.136,Z 415.558,A -85,B 0,C 180,E1 -21608.075,E2 -21608.075} C_VEL
LIN {X 0,Y 199.919,Z 415.583,A -85,B 0,C 180,E1 -21612.177,E2 -21612.177} C_VEL
LIN {X 0,Y 199.81,Z 415.591,A -85,B 0,C 180,E1 -21616.343,E2 -21616.343} C_VEL
LIN {X 0,Y 199.827,Z 415.589,A -85,B 0,C 180,E1 -21618.453,E2 -21618.453} C_VEL
LIN {X 0,Y 199.74,Z 415.604,A -85,B 0,C 180,E1 -21623.817,E2 -21623.817} C_VEL
LIN {X 0,Y 199.716,Z 415.782,A -85,B 0,C 180,E1 -21627.224,E2 -21627.224} C_VEL
LIN {X 0,Y 200.203,Z 418.552,A -85,B 0,C 180,E1 -21631.774,E2 -21631.774} C_VEL
LIN {X 0,Y 200.707,Z 421.785,A -85,B 0,C 180,E1 -21636.532,E2 -21636.532} C_VEL
LIN {X 0,Y 201.137,Z 424.181,A -85,B 0,C 180,E1 -21639.761,E2 -21639.761} C_VEL
LIN {X 0,Y 201.875,Z 427.618,A -85,B 0,C 180,E1 -21644.129,E2 -21644.129} C_VEL
LIN {X 0,Y 202.571,Z 431.574,A -85,B 0,C 180,E1 -21648.762,E2 -21648.762} C_VEL
LIN {X 0,Y 202.76,Z 434.749,A -85,B 0,C 180,E1 -21652.254,E2 -21652.254} C_VEL
LIN {X 0,Y 203.823,Z 438.424,A -85,B 0,C 180,E1 -21652.731,E2 -21652.731} C_VEL
LIN {X 0,Y 206.942,Z 449.743,A -85,B 0,C 180,E1 -21654.265,E2 -21654.265} C_VEL
LIN {X 0,Y 209.182,Z 461.995,A -85,B 0,C 180,E1 -21656.04,E2 -21656.04} C_VEL
LIN {X 0,Y 210.463,Z 473.969,A -85,B 0,C 180,E1 -21657.986,E2 -21657.986} C_VEL
LIN {X 0,Y 210.688,Z 485.66,A -85,B 0,C 180,E1 -21660.146,E2 -21660.146} C_VEL
LIN {X 0,Y 210.134,Z 495.91,A -85,B 0,C 180,E1 -21662.351,E2 -21662.351} C_VEL
LIN {X 0,Y 209.391,Z 501.119,A -85,B 0,C 180,E1 -21663.594,E2 -21663.594} C_VEL
LIN {X 0,Y 206.578,Z 509.986,A -85,B 0,C 180,E1 -21665.904,E2 -21665.904} C_VEL
LIN {X 0,Y 203.894,Z 518.508,A -85,B 0,C 180,E1 -21668.72,E2 -21668.72} C_VEL
LIN {X 0,Y 202.352,Z 523.441,A -85,B 0,C 180,E1 -21670.734,E2 -21670.734} C_VEL
LIN {X 0,Y 200.419,Z 529.302,A -85,B 0,C 180,E1 -21673.62,E2 -21673.62} C_VEL
LIN {X 0,Y 198.932,Z 531.882,A -85,B 0,C 180,E1 -21675.088,E2 -21675.088} C_VEL
LIN {X 0,Y 193.455,Z 536.672,A -85,B 0,C 180,E1 -21678.551,E2 -21678.551} C_VEL
LIN {X 0,Y 191.06,Z 538.724,A -85,B 0,C 180,E1 -21680.719,E2 -21680.719} C_VEL
LIN {X 0,Y 190.598,Z 539.572,A -85,B 0,C 180,E1 -21681.869,E2 -21681.869} C_VEL
LIN {X 0,Y 190.429,Z 541.557,A -85,B 0,C 180,E1 -21685.182,E2 -21685.182} C_VEL
LIN {X 0,Y 190.488,Z 542.415,A -85,B 0,C 180,E1 -21687.885,E2 -21687.885} C_VEL
LIN {X 0,Y 190.607,Z 542.64,A -85,B 0,C 180,E1 -21690,E2 -21690} C_VEL
LIN {X 0,Y 190.493,Z 542.406,A -85,B 0,C 180,E1 -21692.114,E2 -21692.114} C_VEL
LIN {X 0,Y 190.404,Z 541.576,A -85,B 0,C 180,E1 -21694.727,E2 -21694.727} C_VEL
LIN {X 0,Y 190.637,Z 539.306,A -85,B 0,C 180,E1 -21698.48,E2 -21698.48} C_VEL
LIN {X 0,Y 191.285,Z 536.311,A -85,B 0,C 180,E1 -21701.658,E2 -21701.658} C_VEL
LIN {X 0,Y 192.383,Z 532.272,A -85,B 0,C 180,E1 -21704.816,E2 -21704.816} C_VEL
LIN {X 0,Y 194.485,Z 526.093,A -85,B 0,C 180,E1 -21708.433,E2 -21708.433} C_VEL
LIN {X 0,Y 196.795,Z 519.54,A -85,B 0,C 180,E1 -21711.393,E2 -21711.393} C_VEL
LIN {X 0,Y 199.541,Z 511.009,A -85,B 0,C 180,E1 -21714.446,E2 -21714.446} C_VEL
LIN {X 0,Y 202.426,Z 502.472,A -85,B 0,C 180,E1 -21716.83,E2 -21716.83} C_VEL
LIN {X 0,Y 203.383,Z 497.448,A -85,B 0,C 180,E1 -21718.087,E2 -21718.087} C_VEL
LIN {X 0,Y 204.112,Z 486.467,A -85,B 0,C 180,E1 -21720.593,E2 -21720.593} C_VEL
LIN {X 0,Y 204.088,Z 477.14,A -85,B 0,C 180,E1 -21722.443,E2 -21722.443} C_VEL
LIN {X 0,Y 203.34,Z 466.658,A -85,B 0,C 180,E1 -21724.3,E2 -21724.3} C_VEL
LIN {X 0,Y 201.684,Z 455.259,A -85,B 0,C 180,E1 -21726.121,E2 -21726.121} C_VEL
LIN {X 0,Y 198.763,Z 442.787,A -85,B 0,C 180,E1 -21727.968,E2 -21727.968} C_VEL
LIN {X 0,Y 197.136,Z 438.18,A -85,B 0,C 180,E1 -21728.677,E2 -21728.677} C_VEL
LIN {X 0,Y 195.834,Z 434.788,A -85,B 0,C 180,E1 -21729.204,E2 -21729.204} C_VEL
LIN {X 0,Y 195.725,Z 434.214,A -85,B 0,C 180,E1 -21729.292,E2 -21729.292} C_VEL
LIN {X 0,Y 195.241,Z 430.934,A -85,B 0,C 180,E1 -21733.152,E2 -21733.152} C_VEL
LIN {X 0,Y 194.48,Z 427.07,A -85,B 0,C 180,E1 -21738.045,E2 -21738.045} C_VEL
LIN {X 0,Y 193.789,Z 423.51,A -85,B 0,C 180,E1 -21742.926,E2 -21742.926} C_VEL
LIN {X 0,Y 193.353,Z 420.805,A -85,B 0,C 180,E1 -21746.96,E2 -21746.96} C_VEL
LIN {X 0,Y 192.914,Z 417.897,A -85,B 0,C 180,E1 -21751.732,E2 -21751.732} C_VEL
LIN {X 0,Y 192.645,Z 416.489,A -85,B 0,C 180,E1 -21754.529,E2 -21754.529} C_VEL
LIN {X 0,Y 192.639,Z 416.489,A -85,B 0,C 180,E1 -21758.603,E2 -21758.603} C_VEL
LIN {X 0,Y 192.76,Z 416.474,A -85,B 0,C 180,E1 -21763.042,E2 -21763.042} C_VEL
LIN {X 0,Y 192.856,Z 416.463,A -85,B 0,C 180,E1 -21767.37,E2 -21767.37} C_VEL
LIN {X 0,Y 193.082,Z 416.434,A -85,B 0,C 180,E1 -21771.628,E2 -21771.628} C_VEL
LIN {X 0,Y 193.267,Z 416.412,A -85,B 0,C 180,E1 -21777.916,E2 -21777.916} C_VEL
LIN {X 0,Y 193.449,Z 416.388,A -85,B 0,C 180,E1 -21780,E2 -21780} C_VEL
LIN {X 0,Y 192.982,Z 416.445,A -85,B 0,C 180,E1 -21784.177,E2 -21784.177} C_VEL
LIN {X 0,Y 193.082,Z 416.435,A -85,B 0,C 180,E1 -21788.372,E2 -21788.372} C_VEL
LIN {X 0,Y 192.856,Z 416.459,A -85,B 0,C 180,E1 -21792.63,E2 -21792.63} C_VEL
LIN {X 0,Y 192.76,Z 416.474,A -85,B 0,C 180,E1 -21796.959,E2 -21796.959} C_VEL
LIN {X 0,Y 192.624,Z 416.49,A -85,B 0,C 180,E1 -21801.399,E2 -21801.399} C_VEL
LIN {X 0,Y 192.649,Z 416.486,A -85,B 0,C 180,E1 -21804.214,E2 -21804.214} C_VEL
LIN {X 0,Y 192.646,Z 416.487,A -85,B 0,C 180,E1 -21808.889,E2 -21808.889} C_VEL
LIN {X 0,Y 192.6,Z 416.486,A -85,B 0,C 180,E1 -21813.186,E2 -21813.186} C_VEL
LIN {X 0,Y 192.57,Z 416.499,A -85,B 0,C 180,E1 -21818.348,E2 -21818.348} C_VEL
LIN {X 0,Y 192.541,Z 416.498,A -85,B 0,C 180,E1 -21823.111,E2 -21823.111} C_VEL
LIN {X 0,Y 192.601,Z 416.495,A -85,B 0,C 180,E1 -21826.87,E2 -21826.87} C_VEL
LIN {X 0,Y 192.582,Z 416.497,A -85,B 0,C 180,E1 -21828.937,E2 -21828.937} C_VEL
LIN {X 0,Y 192.648,Z 417.103,A -85,B 0,C 180,E1 -21830.099,E2 -21830.099} C_VEL
LIN {X 0,Y 193.849,Z 419.995,A -85,B 0,C 180,E1 -21830.612,E2 -21830.612} C_VEL
LIN {X 0,Y 195.131,Z 421.824,A -85,B 0,C 180,E1 -21831.063,E2 -21831.063} C_VEL
LIN {X 0,Y 199.993,Z 432.016,A -85,B 0,C 180,E1 -21833.164,E2 -21833.164} C_VEL
LIN {X 0,Y 203.972,Z 442.949,A -85,B 0,C 180,E1 -21835.388,E2 -21835.388} C_VEL
LIN {X 0,Y 206.456,Z 452.613,A -85,B 0,C 180,E1 -21837.407,E2 -21837.407} C_VEL
LIN {X 0,Y 208.07,Z 462.309,A -85,B 0,C 180,E1 -21839.559,E2 -21839.559} C_VEL
LIN {X 0,Y 208.482,Z 467.36,A -85,B 0,C 180,E1 -21840.738,E2 -21840.738} C_VEL
LIN {X 0,Y 205.853,Z 477.081,A -85,B 0,C 180,E1 -21842.787,E2 -21842.787} C_VEL
LIN {X 0,Y 202.747,Z 486.989,A -85,B 0,C 180,E1 -21845.42,E2 -21845.42} C_VEL
LIN {X 0,Y 199.699,Z 495.563,A -85,B 0,C 180,E1 -21848.314,E2 -21848.314} C_VEL
LIN {X 0,Y 197.22,Z 502.385,A -85,B 0,C 180,E1 -21851.294,E2 -21851.294} C_VEL
LIN {X 0,Y 195.047,Z 507.849,A -85,B 0,C 180,E1 -21854.321,E2 -21854.321} C_VEL
LIN {X 0,Y 193.416,Z 512.128,A -85,B 0,C 180,E1 -21857.408,E2 -21857.408} C_VEL
LIN {X 0,Y 192.066,Z 515.831,A -85,B 0,C 180,E1 -21861.107,E2 -21861.107} C_VEL
LIN {X 0,Y 191.424,Z 517.602,A -85,B 0,C 180,E1 -21863.677,E2 -21863.677} C_VEL
LIN {X 0,Y 191.064,Z 518.584,A -85,B 0,C 180,E1 -21865.781,E2 -21865.781} C_VEL
LIN {X 0,Y 190.723,Z 519.416,A -85,B 0,C 180,E1 -21870,E2 -21870} C_VEL
LIN {X 0,Y 191.055,Z 518.635,A -85,B 0,C 180,E1 -21874.219,E2 -21874.219} C_VEL
LIN {X 0,Y 191.418,Z 517.674,A -85,B 0,C 180,E1 -21876.324,E2 -21876.324} C_VEL
LIN {X 0,Y 191.946,Z 516.147,A -85,B 0,C 180,E1 -21878.66,E2 -21878.66} C_VEL
LIN {X 0,Y 193.327,Z 512.297,A -85,B 0,C 180,E1 -21882.599,E2 -21882.599} C_VEL
LIN {X 0,Y 195.018,Z 508.065,A -85,B 0,C 180,E1 -21885.681,E2 -21885.681} C_VEL
LIN {X 0,Y 197.533,Z 501.654,A -85,B 0,C 180,E1 -21889.215,E2 -21889.215} C_VEL
LIN {X 0,Y 200.107,Z 494.603,A -85,B 0,C 180,E1 -21892.183,E2 -21892.183} C_VEL
LIN {X 0,Y 203.304,Z 485.802,A -85,B 0,C 180,E1 -21895.054,E2 -21895.054} C_VEL
LIN {X 0,Y 206.05,Z 476.663,A -85,B 0,C 180,E1 -21897.451,E2 -21897.451} C_VEL
LIN {X 0,Y 208.582,Z 466.779,A -85,B 0,C 180,E1 -21899.524,E2 -21899.524} C_VEL
LIN {X 0,Y 207.383,Z 457.2,A -85,B 0,C 180,E1 -21901.735,E2 -21901.735} C_VEL
LIN {X 0,Y 205.387,Z 447.893,A -85,B 0,C 180,E1 -21903.74,E2 -21903.74} C_VEL
LIN {X 0,Y 202.396,Z 437.886,A -85,B 0,C 180,E1 -21905.783,E2 -21905.783} C_VEL
LIN {X 0,Y 198.214,Z 428.149,A -85,B 0,C 180,E1 -21907.812,E2 -21907.812} C_VEL
LIN {X 0,Y 194.474,Z 420.882,A -85,B 0,C 180,E1 -21909.336,E2 -21909.336} C_VEL
LIN {X 0,Y 192.942,Z 418.306,A -85,B 0,C 180,E1 -21909.912,E2 -21909.912} C_VEL
LIN {X 0,Y 192.588,Z 416.978,A -85,B 0,C 180,E1 -21910.138,E2 -21910.138} C_VEL
LIN {X 0,Y 192.527,Z 416.558,A -85,B 0,C 180,E1 -21911.078,E2 -21911.078} C_VEL
LIN {X 0,Y 192.516,Z 416.503,A -85,B 0,C 180,E1 -21916.083,E2 -21916.083} C_VEL
LIN {X 0,Y 192.544,Z 416.5,A -85,B 0,C 180,E1 -21920.043,E2 -21920.043} C_VEL
LIN {X 0,Y 192.601,Z 416.488,A -85,B 0,C 180,E1 -21924.279,E2 -21924.279} C_VEL
LIN {X 0,Y 192.603,Z 416.493,A -85,B 0,C 180,E1 -21929.279,E2 -21929.279} C_VEL
LIN {X 0,Y 192.664,Z 416.487,A -85,B 0,C 180,E1 -21931.691,E2 -21931.691} C_VEL
LIN {X 0,Y 192.688,Z 416.484,A -85,B 0,C 180,E1 -21936.346,E2 -21936.346} C_VEL
LIN {X 0,Y 192.735,Z 416.476,A -85,B 0,C 180,E1 -21941.458,E2 -21941.458} C_VEL
LIN {X 0,Y 192.775,Z 416.472,A -85,B 0,C 180,E1 -21945.214,E2 -21945.214} C_VEL
LIN {X 0,Y 192.948,Z 416.449,A -85,B 0,C 180,E1 -21949.567,E2 -21949.567} C_VEL
LIN {X 0,Y 192.986,Z 416.449,A -85,B 0,C 180,E1 -21953.728,E2 -21953.728} C_VEL
LIN {X 0,Y 193.266,Z 416.413,A -85,B 0,C 180,E1 -21957.916,E2 -21957.916} C_VEL
LIN {X 0,Y 193.447,Z 416.393,A -85,B 0,C 180,E1 -21960,E2 -21960} C_VEL
LIN {X 0,Y 192.984,Z 416.449,A -85,B 0,C 180,E1 -21964.177,E2 -21964.177} C_VEL
LIN {X 0,Y 193.083,Z 416.436,A -85,B 0,C 180,E1 -21968.372,E2 -21968.372} C_VEL
LIN {X 0,Y 192.857,Z 416.462,A -85,B 0,C 180,E1 -21972.63,E2 -21972.63} C_VEL
LIN {X 0,Y 192.784,Z 416.467,A -85,B 0,C 180,E1 -21978.586,E2 -21978.586} C_VEL
LIN {X 0,Y 192.667,Z 416.486,A -85,B 0,C 180,E1 -21984.225,E2 -21984.225} C_VEL
LIN {X 0,Y 192.682,Z 416.69,A -85,B 0,C 180,E1 -21985.957,E2 -21985.957} C_VEL
LIN {X 0,Y 193.007,Z 418.42,A -85,B 0,C 180,E1 -21989.082,E2 -21989.082} C_VEL
LIN {X 0,Y 193.389,Z 421.029,A -85,B 0,C 180,E1 -21993.295,E2 -21993.295} C_VEL
LIN {X 0,Y 193.908,Z 424.246,A -85,B 0,C 180,E1 -21998.035,E2 -21998.035} C_VEL
LIN {X 0,Y 194.836,Z 428.57,A -85,B 0,C 180,E1 -22003.827,E2 -22003.827} C_VEL
LIN {X 0,Y 195.258,Z 431.006,A -85,B 0,C 180,E1 -22006.852,E2 -22006.852} C_VEL
LIN {X 0,Y 195.718,Z 434.279,A -85,B 0,C 180,E1 -22010.671,E2 -22010.671} C_VEL
LIN {X 0,Y 196.762,Z 437.546,A -85,B 0,C 180,E1 -22011.124,E2 -22011.124} C_VEL
LIN {X 0,Y 197.728,Z 439.71,A -85,B 0,C 180,E1 -22011.497,E2 -22011.497} C_VEL
LIN {X 0,Y 200.343,Z 448.85,A -85,B 0,C 180,E1 -22012.854,E2 -22012.854} C_VEL
LIN {X 0,Y 202.577,Z 460.32,A -85,B 0,C 180,E1 -22014.614,E2 -22014.614} C_VEL
LIN {X 0,Y 203.835,Z 471.697,A -85,B 0,C 180,E1 -22016.518,E2 -22016.518} C_VEL
LIN {X 0,Y 204.27,Z 483.016,A -85,B 0,C 180,E1 -22018.658,E2 -22018.658} C_VEL
LIN {X 0,Y 203.85,Z 492.757,A -85,B 0,C 180,E1 -22020.747,E2 -22020.747} C_VEL
LIN {X 0,Y 202.937,Z 500.682,A -85,B 0,C 180,E1 -22022.686,E2 -22022.686} C_VEL
LIN {X 0,Y 200.075,Z 509.553,A -85,B 0,C 180,E1 -22025.069,E2 -22025.069} C_VEL
LIN {X 0,Y 197.404,Z 517.561,A -85,B 0,C 180,E1 -22027.768,E2 -22027.768} C_VEL
LIN {X 0,Y 195.656,Z 523.01,A -85,B 0,C 180,E1 -22030.047,E2 -22030.047} C_VEL
LIN {X 0,Y 193.438,Z 529.282,A -85,B 0,C 180,E1 -22033.267,E2 -22033.267} C_VEL
LIN {X 0,Y 191.97,Z 533.787,A -85,B 0,C 180,E1 -22036.233,E2 -22036.233} C_VEL
LIN {X 0,Y 191.037,Z 537.446,A -85,B 0,C 180,E1 -22039.4,E2 -22039.4} C_VEL
LIN {X 0,Y 190.598,Z 539.572,A -85,B 0,C 180,E1 -22041.869,E2 -22041.869} C_VEL
LIN {X 0,Y 189.819,Z 540.719,A -85,B 0,C 180,E1 -22043.604,E2 -22043.604} C_VEL
LIN {X 0,Y 188.225,Z 541.512,A -85,B 0,C 180,E1 -22045.324,E2 -22045.324} C_VEL
LIN {X 0,Y 184.585,Z 542.193,A -85,B 0,C 180,E1 -22048.832,E2 -22048.832} C_VEL
LIN {X 0,Y 183.535,Z 542.165,A -85,B 0,C 180,E1 -22050.669,E2 -22050.669} C_VEL
LIN {X 0,Y 183.429,Z 542.071,A -85,B 0,C 180,E1 -22051.291,E2 -22051.291} C_VEL
LIN {X 0,Y 183.33,Z 541.244,A -85,B 0,C 180,E1 -22054.644,E2 -22054.644} C_VEL
LIN {X 0,Y 183.584,Z 538.871,A -85,B 0,C 180,E1 -22058.808,E2 -22058.808} C_VEL
LIN {X 0,Y 184.311,Z 535.876,A -85,B 0,C 180,E1 -22062.106,E2 -22062.106} C_VEL
LIN {X 0,Y 185.489,Z 531.836,A -85,B 0,C 180,E1 -22065.38,E2 -22065.38} C_VEL
LIN {X 0,Y 187.694,Z 525.655,A -85,B 0,C 180,E1 -22069.125,E2 -22069.125} C_VEL
LIN {X 0,Y 189.796,Z 520.17,A -85,B 0,C 180,E1 -22071.734,E2 -22071.734} C_VEL
LIN {X 0,Y 192.518,Z 512.07,A -85,B 0,C 180,E1 -22074.823,E2 -22074.823} C_VEL
LIN {X 0,Y 195.451,Z 503.845,A -85,B 0,C 180,E1 -22077.288,E2 -22077.288} C_VEL
LIN {X 0,Y 196.493,Z 500.059,A -85,B 0,C 180,E1 -22078.289,E2 -22078.289} C_VEL
LIN {X 0,Y 197.522,Z 489.511,A -85,B 0,C 180,E1 -22080.921,E2 -22080.921} C_VEL
LIN {X 0,Y 197.77,Z 480.024,A -85,B 0,C 180,E1 -22082.964,E2 -22082.964} C_VEL
LIN {X 0,Y 197.181,Z 468.354,A -85,B 0,C 180,E1 -22085.196,E2 -22085.196} C_VEL
LIN {X 0,Y 195.845,Z 457.791,A -85,B 0,C 180,E1 -22087.012,E2 -22087.012} C_VEL
LIN {X 0,Y 193.079,Z 445.285,A -85,B 0,C 180,E1 -22089.029,E2 -22089.029} C_VEL
LIN {X 0,Y 191.629,Z 441.23,A -85,B 0,C 180,E1 -22089.742,E2 -22089.742} C_VEL
LIN {X 0,Y 190.15,Z 437.815,A -85,B 0,C 180,E1 -22090.367,E2 -22090.367} C_VEL
LIN {X 0,Y 188.712,Z 434.484,A -85,B 0,C 180,E1 -22090.974,E2 -22090.974} C_VEL
LIN {X 0,Y 188.551,Z 433.688,A -85,B 0,C 180,E1 -22091.066,E2 -22091.066} C_VEL
LIN {X 0,Y 187.882,Z 430.368,A -85,B 0,C 180,E1 -22095.294,E2 -22095.294} C_VEL
LIN {X 0,Y 187.397,Z 427.918,A -85,B 0,C 180,E1 -22098.596,E2 -22098.596} C_VEL
LIN {X 0,Y 186.839,Z 424.842,A -85,B 0,C 180,E1 -22102.998,E2 -22102.998} C_VEL
LIN {X 0,Y 186.265,Z 421.573,A -85,B 0,C 180,E1 -22108.114,E2 -22108.114} C_VEL
LIN {X 0,Y 186.082,Z 420.105,A -85,B 0,C 180,E1 -22110.594,E2 -22110.594} C_VEL
LIN {X 0,Y 185.634,Z 417.362,A -85,B 0,C 180,E1 -22115.984,E2 -22115.984} C_VEL
LIN {X 0,Y 185.677,Z 417.356,A -85,B 0,C 180,E1 -22121.133,E2 -22121.133} C_VEL
LIN {X 0,Y 185.727,Z 417.351,A -85,B 0,C 180,E1 -22124.64,E2 -22124.64} C_VEL
LIN {X 0,Y 185.945,Z 417.324,A -85,B 0,C 180,E1 -22129.328,E2 -22129.328} C_VEL
LIN {X 0,Y 185.972,Z 417.321,A -85,B 0,C 180,E1 -22133.49,E2 -22133.49} C_VEL
LIN {X 0,Y 186.211,Z 417.291,A -85,B 0,C 180,E1 -22137.837,E2 -22137.837} C_VEL
LIN {X 0,Y 186.412,Z 417.265,A -85,B 0,C 180,E1 -22140,E2 -22140} C_VEL
LIN {X 0,Y 185.93,Z 417.323,A -85,B 0,C 180,E1 -22144.336,E2 -22144.336} C_VEL
LIN {X 0,Y 186.032,Z 417.312,A -85,B 0,C 180,E1 -22148.692,E2 -22148.692} C_VEL
LIN {X 0,Y 185.767,Z 417.342,A -85,B 0,C 180,E1 -22153.12,E2 -22153.12} C_VEL
LIN {X 0,Y 185.692,Z 417.355,A -85,B 0,C 180,E1 -22157.625,E2 -22157.625} C_VEL
LIN {X 0,Y 185.583,Z 417.367,A -85,B 0,C 180,E1 -22162.253,E2 -22162.253} C_VEL
LIN {X 0,Y 185.56,Z 417.368,A -85,B 0,C 180,E1 -22167.033,E2 -22167.033} C_VEL
LIN {X 0,Y 185.579,Z 417.367,A -85,B 0,C 180,E1 -22169.493,E2 -22169.493} C_VEL
LIN {X 0,Y 185.511,Z 417.377,A -85,B 0,C 180,E1 -22174.63,E2 -22174.63} C_VEL
LIN {X 0,Y 185.528,Z 417.37,A -85,B 0,C 180,E1 -22177.308,E2 -22177.308} C_VEL
LIN {X 0,Y 185.496,Z 417.376,A -85,B 0,C 180,E1 -22180.733,E2 -22180.733} C_VEL
LIN {X 0,Y 185.556,Z 417.372,A -85,B 0,C 180,E1 -22186.025,E2 -22186.025} C_VEL
LIN {X 0,Y 185.537,Z 417.505,A -85,B 0,C 180,E1 -22188.186,E2 -22188.186} C_VEL
LIN {X 0,Y 186.681,Z 420.448,A -85,B 0,C 180,E1 -22188.771,E2 -22188.771} C_VEL
LIN {X 0,Y 188.337,Z 422.905,A -85,B 0,C 180,E1 -22189.414,E2 -22189.414} C_VEL
LIN {X 0,Y 192.146,Z 430.171,A -85,B 0,C 180,E1 -22191.115,E2 -22191.115} C_VEL
LIN {X 0,Y 195.921,Z 439.178,A -85,B 0,C 180,E1 -22193.115,E2 -22193.115} C_VEL
LIN {X 0,Y 198.897,Z 448.837,A -85,B 0,C 180,E1 -22195.239,E2 -22195.239} C_VEL
LIN {X 0,Y 200.981,Z 458.72,A -85,B 0,C 180,E1 -22197.494,E2 -22197.494} C_VEL
LIN {X 0,Y 202.085,Z 467.813,A -85,B 0,C 180,E1 -22199.717,E2 -22199.717} C_VEL
LIN {X 0,Y 201.331,Z 471.305,A -85,B 0,C 180,E1 -22200.457,E2 -22200.457} C_VEL
LIN {X 0,Y 198.667,Z 480.566,A -85,B 0,C 180,E1 -22202.62,E2 -22202.62} C_VEL
LIN {X 0,Y 195.771,Z 489.009,A -85,B 0,C 180,E1 -22205.051,E2 -22205.051} C_VEL
LIN {X 0,Y 192.677,Z 497.215,A -85,B 0,C 180,E1 -22208.045,E2 -22208.045} C_VEL
LIN {X 0,Y 190.514,Z 502.818,A -85,B 0,C 180,E1 -22210.609,E2 -22210.609} C_VEL
LIN {X 0,Y 188.252,Z 508.281,A -85,B 0,C 180,E1 -22213.74,E2 -22213.74} C_VEL
LIN {X 0,Y 186.493,Z 512.561,A -85,B 0,C 180,E1 -22216.932,E2 -22216.932} C_VEL
LIN {X 0,Y 184.988,Z 516.481,A -85,B 0,C 180,E1 -22221.036,E2 -22221.036} C_VEL
LIN {X 0,Y 184.385,Z 518.034,A -85,B 0,C 180,E1 -22223.434,E2 -22223.434} C_VEL
LIN {X 0,Y 184.019,Z 519.014,A -85,B 0,C 180,E1 -22225.619,E2 -22225.619} C_VEL
LIN {X 0,Y 183.657,Z 519.846,A -85,B 0,C 180,E1 -22230,E2 -22230} C_VEL
LIN {X 0,Y 184.01,Z 519.065,A -85,B 0,C 180,E1 -22234.381,E2 -22234.381} C_VEL
LIN {X 0,Y 184.379,Z 518.105,A -85,B 0,C 180,E1 -22236.566,E2 -22236.566} C_VEL
LIN {X 0,Y 184.879,Z 516.76,A -85,B 0,C 180,E1 -22238.746,E2 -22238.746} C_VEL
LIN {X 0,Y 185.962,Z 513.916,A -85,B 0,C 180,E1 -22241.997,E2 -22241.997} C_VEL
LIN {X 0,Y 187.558,Z 510.048,A -85,B 0,C 180,E1 -22245.207,E2 -22245.207} C_VEL
LIN {X 0,Y 189.619,Z 505.054,A -85,B 0,C 180,E1 -22248.364,E2 -22248.364} C_VEL
LIN {X 0,Y 192.167,Z 498.756,A -85,B 0,C 180,E1 -22251.452,E2 -22251.452} C_VEL
LIN {X 0,Y 195.204,Z 490.869,A -85,B 0,C 180,E1 -22254.459,E2 -22254.459} C_VEL
LIN {X 0,Y 198.046,Z 482.825,A -85,B 0,C 180,E1 -22256.902,E2 -22256.902} C_VEL
LIN {X 0,Y 200.926,Z 473.019,A -85,B 0,C 180,E1 -22259.321,E2 -22259.321} C_VEL
LIN {X 0,Y 202.158,Z 468.427,A -85,B 0,C 180,E1 -22260.272,E2 -22260.272} C_VEL
LIN {X 0,Y 201.058,Z 458.616,A -85,B 0,C 180,E1 -22262.667,E2 -22262.667} C_VEL
LIN {X 0,Y 198.71,Z 447.812,A -85,B 0,C 180,E1 -22265.126,E2 -22265.126} C_VEL
LIN {X 0,Y 195.695,Z 438.359,A -85,B 0,C 180,E1 -22267.213,E2 -22267.213} C_VEL
LIN {X 0,Y 190.791,Z 427.448,A -85,B 0,C 180,E1 -22269.688,E2 -22269.688} C_VEL
LIN {X 0,Y 188.072,Z 422.398,A -85,B 0,C 180,E1 -22270.873,E2 -22270.873} C_VEL
LIN {X 0,Y 185.89,Z 419.133,A -85,B 0,C 180,E1 -22271.733,E2 -22271.733} C_VEL
LIN {X 0,Y 185.479,Z 417.526,A -85,B 0,C 180,E1 -22272.007,E2 -22272.007} C_VEL
LIN {X 0,Y 185.48,Z 417.381,A -85,B 0,C 180,E1 -22276.997,E2 -22276.997} C_VEL
LIN {X 0,Y 185.493,Z 417.379,A -85,B 0,C 180,E1 -22279.901,E2 -22279.901} C_VEL
LIN {X 0,Y 185.546,Z 417.374,A -85,B 0,C 180,E1 -22282.696,E2 -22282.696} C_VEL
LIN {X 0,Y 185.544,Z 417.372,A -85,B 0,C 180,E1 -22287.975,E2 -22287.975} C_VEL
LIN {X 0,Y 185.583,Z 417.368,A -85,B 0,C 180,E1 -22290.577,E2 -22290.577} C_VEL
LIN {X 0,Y 185.583,Z 417.365,A -85,B 0,C 180,E1 -22295.382,E2 -22295.382} C_VEL
LIN {X 0,Y 185.677,Z 417.354,A -85,B 0,C 180,E1 -22301.133,E2 -22301.133} C_VEL
LIN {X 0,Y 185.728,Z 417.35,A -85,B 0,C 180,E1 -22304.64,E2 -22304.64} C_VEL
LIN {X 0,Y 185.891,Z 417.328,A -85,B 0,C 180,E1 -22309.418,E2 -22309.418} C_VEL
LIN {X 0,Y 185.949,Z 417.324,A -85,B 0,C 180,E1 -22313.489,E2 -22313.489} C_VEL
LIN {X 0,Y 186.21,Z 417.292,A -85,B 0,C 180,E1 -22317.837,E2 -22317.837} C_VEL
LIN {X 0,Y 186.411,Z 417.269,A -85,B 0,C 180,E1 -22320,E2 -22320} C_VEL
LIN {X 0,Y 185.931,Z 417.328,A -85,B 0,C 180,E1 -22324.335,E2 -22324.335} C_VEL
LIN {X 0,Y 186.033,Z 417.314,A -85,B 0,C 180,E1 -22328.691,E2 -22328.691} C_VEL
LIN {X 0,Y 185.769,Z 417.346,A -85,B 0,C 180,E1 -22333.12,E2 -22333.12} C_VEL
LIN {X 0,Y 185.72,Z 417.341,A -85,B 0,C 180,E1 -22337.622,E2 -22337.622} C_VEL
LIN {X 0,Y 185.635,Z 417.362,A -85,B 0,C 180,E1 -22344.016,E2 -22344.016} C_VEL
LIN {X 0,Y 186.085,Z 420.165,A -85,B 0,C 180,E1 -22349.405,E2 -22349.405} C_VEL
LIN {X 0,Y 186.514,Z 423.211,A -85,B 0,C 180,E1 -22354.417,E2 -22354.417} C_VEL
LIN {X 0,Y 186.923,Z 425.476,A -85,B 0,C 180,E1 -22357.854,E2 -22357.854} C_VEL
LIN {X 0,Y 187.582,Z 428.709,A -85,B 0,C 180,E1 -22362.407,E2 -22362.407} C_VEL
LIN {X 0,Y 188.211,Z 431.84,A -85,B 0,C 180,E1 -22366.508,E2 -22366.508} C_VEL
LIN {X 0,Y 188.543,Z 433.737,A -85,B 0,C 180,E1 -22368.861,E2 -22368.861} C_VEL
LIN {X 0,Y 189.639,Z 436.947,A -85,B 0,C 180,E1 -22369.363,E2 -22369.363} C_VEL
LIN {X 0,Y 190.95,Z 439.478,A -85,B 0,C 180,E1 -22369.882,E2 -22369.882} C_VEL
LIN {X 0,Y 193.39,Z 446.312,A -85,B 0,C 180,E1 -22371.066,E2 -22371.066} C_VEL
LIN {X 0,Y 195.922,Z 458.167,A -85,B 0,C 180,E1 -22372.988,E2 -22372.988} C_VEL
LIN {X 0,Y 197.344,Z 469.672,A -85,B 0,C 180,E1 -22374.995,E2 -22374.995} C_VEL
LIN {X 0,Y 197.81,Z 480.246,A -85,B 0,C 180,E1 -22377.032,E2 -22377.032} C_VEL
LIN {X 0,Y 197.478,Z 491.21,A -85,B 0,C 180,E1 -22379.435,E2 -22379.435} C_VEL
LIN {X 0,Y 196.494,Z 500.241,A -85,B 0,C 180,E1 -22381.711,E2 -22381.711} C_VEL
LIN {X 0,Y 194.238,Z 507.484,A -85,B 0,C 180,E1 -22383.689,E2 -22383.689} C_VEL
LIN {X 0,Y 191.161,Z 516.109,A -85,B 0,C 180,E1 -22386.574,E2 -22386.574} C_VEL
LIN {X 0,Y 188.99,Z 522.579,A -85,B 0,C 180,E1 -22389.312,E2 -22389.312} C_VEL
LIN {X 0,Y 186.724,Z 528.591,A -85,B 0,C 180,E1 -22392.475,E2 -22392.475} C_VEL
LIN {X 0,Y 185.022,Z 533.352,A -85,B 0,C 180,E1 -22395.706,E2 -22395.706} C_VEL
LIN {X 0,Y 184.037,Z 537.013,A -85,B 0,C 180,E1 -22398.992,E2 -22398.992} C_VEL
LIN {X 0,Y 183.509,Z 539.307,A -85,B 0,C 180,E1 -22401.814,E2 -22401.814} C_VEL
LIN {X 0,Y 183.337,Z 541.354,A -85,B 0,C 180,E1 -22405.603,E2 -22405.603} C_VEL
LIN {X 0,Y 183.402,Z 541.983,A -85,B 0,C 180,E1 -22407.804,E2 -22407.804} C_VEL
LIN {X 0,Y 183.541,Z 542.21,A -85,B 0,C 180,E1 -22410,E2 -22410} C_VEL
LIN {X 0,Y 183.429,Z 542.071,A -85,B 0,C 180,E1 -22411.291,E2 -22411.291} C_VEL
LIN {X 0,Y 183.061,Z 541.882,A -85,B 0,C 180,E1 -22412.513,E2 -22412.513} C_VEL
LIN {X 0,Y 181.672,Z 541.306,A -85,B 0,C 180,E1 -22414.313,E2 -22414.313} C_VEL
LIN {X 0,Y 177.58,Z 538.908,A -85,B 0,C 180,E1 -22418.504,E2 -22418.504} C_VEL
LIN {X 0,Y 176.847,Z 537.483,A -85,B 0,C 180,E1 -22420.361,E2 -22420.361} C_VEL
LIN {X 0,Y 176.906,Z 536.921,A -85,B 0,C 180,E1 -22420.984,E2 -22420.984} C_VEL
LIN {X 0,Y 178.103,Z 532.851,A -85,B 0,C 180,E1 -22424.862,E2 -22424.862} C_VEL
LIN {X 0,Y 179.935,Z 528.072,A -85,B 0,C 180,E1 -22428.208,E2 -22428.208} C_VEL
LIN {X 0,Y 182.334,Z 522.042,A -85,B 0,C 180,E1 -22431.48,E2 -22431.48} C_VEL
LIN {X 0,Y 185.02,Z 514.528,A -85,B 0,C 180,E1 -22434.698,E2 -22434.698} C_VEL
LIN {X 0,Y 187.843,Z 506.894,A -85,B 0,C 180,E1 -22437.279,E2 -22437.279} C_VEL
LIN {X 0,Y 189.689,Z 501.589,A -85,B 0,C 180,E1 -22438.793,E2 -22438.793} C_VEL
LIN {X 0,Y 190.922,Z 491.781,A -85,B 0,C 180,E1 -22441.409,E2 -22441.409} C_VEL
LIN {X 0,Y 191.407,Z 482.128,A -85,B 0,C 180,E1 -22443.65,E2 -22443.65} C_VEL
LIN {X 0,Y 191.034,Z 470.399,A -85,B 0,C 180,E1 -22446.06,E2 -22446.06} C_VEL
LIN {X 0,Y 189.845,Z 459.566,A -85,B 0,C 180,E1 -22448.064,E2 -22448.064} C_VEL
LIN {X 0,Y 187.484,Z 447.984,A -85,B 0,C 180,E1 -22450.096,E2 -22450.096} C_VEL
LIN {X 0,Y 185.179,Z 441.909,A -85,B 0,C 180,E1 -22451.305,E2 -22451.305} C_VEL
LIN {X 0,Y 183.299,Z 437.879,A -85,B 0,C 180,E1 -22452.162,E2 -22452.162} C_VEL
LIN {X 0,Y 181.553,Z 434.642,A -85,B 0,C 180,E1 -22452.914,E2 -22452.914} C_VEL
LIN {X 0,Y 181.16,Z 433.098,A -85,B 0,C 180,E1 -22453.175,E2 -22453.175} C_VEL
LIN {X 0,Y 180.44,Z 429.184,A -85,B 0,C 180,E1 -22458.537,E2 -22458.537} C_VEL
LIN {X 0,Y 179.703,Z 425.511,A -85,B 0,C 180,E1 -22464.081,E2 -22464.081} C_VEL
LIN {X 0,Y 179.191,Z 422.168,A -85,B 0,C 180,E1 -22469.639,E2 -22469.639} C_VEL
LIN {X 0,Y 178.754,Z 419.483,A -85,B 0,C 180,E1 -22474.727,E2 -22474.727} C_VEL
LIN {X 0,Y 178.568,Z 418.241,A -85,B 0,C 180,E1 -22477.435,E2 -22477.435} C_VEL
LIN {X 0,Y 178.652,Z 418.232,A -85,B 0,C 180,E1 -22481.657,E2 -22481.657} C_VEL
LIN {X 0,Y 178.69,Z 418.229,A -85,B 0,C 180,E1 -22486.35,E2 -22486.35} C_VEL
LIN {X 0,Y 178.981,Z 418.192,A -85,B 0,C 180,E1 -22490.963,E2 -22490.963} C_VEL
LIN {X 0,Y 179.157,Z 418.169,A -85,B 0,C 180,E1 -22497.752,E2 -22497.752} C_VEL
LIN {X 0,Y 179.375,Z 418.141,A -85,B 0,C 180,E1 -22500,E2 -22500} C_VEL
LIN {X 0,Y 178.878,Z 418.201,A -85,B 0,C 180,E1 -22504.507,E2 -22504.507} C_VEL
LIN {X 0,Y 178.981,Z 418.19,A -85,B 0,C 180,E1 -22509.037,E2 -22509.037} C_VEL
LIN {X 0,Y 178.69,Z 418.224,A -85,B 0,C 180,E1 -22513.65,E2 -22513.65} C_VEL
LIN {X 0,Y 178.651,Z 418.229,A -85,B 0,C 180,E1 -22518.344,E2 -22518.344} C_VEL
LIN {X 0,Y 178.501,Z 418.25,A -85,B 0,C 180,E1 -22523.187,E2 -22523.187} C_VEL
LIN {X 0,Y 178.487,Z 418.253,A -85,B 0,C 180,E1 -22528.197,E2 -22528.197} C_VEL
LIN {X 0,Y 178.478,Z 418.253,A -85,B 0,C 180,E1 -22530.791,E2 -22530.791} C_VEL
LIN {X 0,Y 178.492,Z 418.25,A -85,B 0,C 180,E1 -22534.222,E2 -22534.222} C_VEL
LIN {X 0,Y 178.419,Z 418.26,A -85,B 0,C 180,E1 -22539.069,E2 -22539.069} C_VEL
LIN {X 0,Y 178.426,Z 418.259,A -85,B 0,C 180,E1 -22542.037,E2 -22542.037} C_VEL
LIN {X 0,Y 178.508,Z 418.26,A -85,B 0,C 180,E1 -22546.186,E2 -22546.186} C_VEL
LIN {X 0,Y 179.507,Z 421.049,A -85,B 0,C 180,E1 -22546.731,E2 -22546.731} C_VEL
LIN {X 0,Y 181.415,Z 423.632,A -85,B 0,C 180,E1 -22547.526,E2 -22547.526} C_VEL
LIN {X 0,Y 185.847,Z 431.735,A -85,B 0,C 180,E1 -22549.656,E2 -22549.656} C_VEL
LIN {X 0,Y 190.239,Z 442.358,A -85,B 0,C 180,E1 -22552.233,E2 -22552.233} C_VEL
LIN {X 0,Y 193.028,Z 451.92,A -85,B 0,C 180,E1 -22554.508,E2 -22554.508} C_VEL
LIN {X 0,Y 194.914,Z 462.038,A -85,B 0,C 180,E1 -22556.988,E2 -22556.988} C_VEL
LIN {X 0,Y 195.69,Z 469.423,A -85,B 0,C 180,E1 -22558.918,E2 -22558.918} C_VEL
LIN {X 0,Y 193.085,Z 478.799,A -85,B 0,C 180,E1 -22561.083,E2 -22561.083} C_VEL
LIN {X 0,Y 189.983,Z 487.855,A -85,B 0,C 180,E1 -22563.646,E2 -22563.646} C_VEL
LIN {X 0,Y 186.593,Z 496.431,A -85,B 0,C 180,E1 -22566.704,E2 -22566.704} C_VEL
LIN {X 0,Y 183.839,Z 503.252,A -85,B 0,C 180,E1 -22569.876,E2 -22569.876} C_VEL
LIN {X 0,Y 181.45,Z 508.715,A -85,B 0,C 180,E1 -22573.113,E2 -22573.113} C_VEL
LIN {X 0,Y 179.583,Z 512.995,A -85,B 0,C 180,E1 -22576.42,E2 -22576.42} C_VEL
LIN {X 0,Y 178.631,Z 515.255,A -85,B 0,C 180,E1 -22578.655,E2 -22578.655} C_VEL
LIN {X 0,Y 177.936,Z 517.087,A -85,B 0,C 180,E1 -22580.91,E2 -22580.91} C_VEL
LIN {X 0,Y 177.353,Z 518.466,A -85,B 0,C 180,E1 -22583.173,E2 -22583.173} C_VEL
LIN {X 0,Y 176.976,Z 519.445,A -85,B 0,C 180,E1 -22585.445,E2 -22585.445} C_VEL
LIN {X 0,Y 176.592,Z 520.276,A -85,B 0,C 180,E1 -22590,E2 -22590} C_VEL
LIN {X 0,Y 176.968,Z 519.495,A -85,B 0,C 180,E1 -22594.556,E2 -22594.556} C_VEL
LIN {X 0,Y 177.875,Z 517.191,A -85,B 0,C 180,E1 -22599.094,E2 -22599.094} C_VEL
LIN {X 0,Y 179.021,Z 514.347,A -85,B 0,C 180,E1 -22602.47,E2 -22602.47} C_VEL
LIN {X 0,Y 180.718,Z 510.479,A -85,B 0,C 180,E1 -22605.797,E2 -22605.797} C_VEL
LIN {X 0,Y 182.912,Z 505.484,A -85,B 0,C 180,E1 -22609.063,E2 -22609.063} C_VEL
LIN {X 0,Y 185.575,Z 499.186,A -85,B 0,C 180,E1 -22612.254,E2 -22612.254} C_VEL
LIN {X 0,Y 188.799,Z 491.297,A -85,B 0,C 180,E1 -22615.347,E2 -22615.347} C_VEL
LIN {X 0,Y 191.76,Z 483.253,A -85,B 0,C 180,E1 -22617.859,E2 -22617.859} C_VEL
LIN {X 0,Y 194.781,Z 473.447,A -85,B 0,C 180,E1 -22620.341,E2 -22620.341} C_VEL
LIN {X 0,Y 195.756,Z 470.018,A -85,B 0,C 180,E1 -22621.071,E2 -22621.071} C_VEL
LIN {X 0,Y 194.735,Z 460.128,A -85,B 0,C 180,E1 -22623.635,E2 -22623.635} C_VEL
LIN {X 0,Y 192.589,Z 449.775,A -85,B 0,C 180,E1 -22626.158,E2 -22626.158} C_VEL
LIN {X 0,Y 189.959,Z 441.308,A -85,B 0,C 180,E1 -22628.166,E2 -22628.166} C_VEL
LIN {X 0,Y 185.295,Z 430.612,A -85,B 0,C 180,E1 -22630.808,E2 -22630.808} C_VEL
LIN {X 0,Y 182.733,Z 426.161,A -85,B 0,C 180,E1 -22632.014,E2 -22632.014} C_VEL
LIN {X 0,Y 180.618,Z 422.541,A -85,B 0,C 180,E1 -22632.99,E2 -22632.99} C_VEL
LIN {X 0,Y 178.943,Z 420.203,A -85,B 0,C 180,E1 -22633.705,E2 -22633.705} C_VEL
LIN {X 0,Y 178.414,Z 418.262,A -85,B 0,C 180,E1 -22634.036,E2 -22634.036} C_VEL
LIN {X 0,Y 178.418,Z 418.257,A -85,B 0,C 180,E1 -22638.455,E2 -22638.455} C_VEL
LIN {X 0,Y 178.467,Z 418.251,A -85,B 0,C 180,E1 -22641.963,E2 -22641.963} C_VEL
LIN {X 0,Y 178.492,Z 418.253,A -85,B 0,C 180,E1 -22646.548,E2 -22646.548} C_VEL
LIN {X 0,Y 178.524,Z 418.246,A -85,B 0,C 180,E1 -22650.007,E2 -22650.007} C_VEL
LIN {X 0,Y 178.522,Z 418.245,A -85,B 0,C 180,E1 -22654.886,E2 -22654.886} C_VEL
LIN {X 0,Y 178.625,Z 418.232,A -85,B 0,C 180,E1 -22660.785,E2 -22660.785} C_VEL
LIN {X 0,Y 178.669,Z 418.228,A -85,B 0,C 180,E1 -22664.017,E2 -22664.017} C_VEL
LIN {X 0,Y 178.837,Z 418.206,A -85,B 0,C 180,E1 -22669.256,E2 -22669.256} C_VEL
LIN {X 0,Y 178.912,Z 418.199,A -85,B 0,C 180,E1 -22673.232,E2 -22673.232} C_VEL
LIN {X 0,Y 179.156,Z 418.171,A -85,B 0,C 180,E1 -22677.752,E2 -22677.752} C_VEL
LIN {X 0,Y 179.374,Z 418.146,A -85,B 0,C 180,E1 -22680,E2 -22680} C_VEL
LIN {X 0,Y 178.88,Z 418.206,A -85,B 0,C 180,E1 -22684.507,E2 -22684.507} C_VEL
LIN {X 0,Y 178.982,Z 418.191,A -85,B 0,C 180,E1 -22689.037,E2 -22689.037} C_VEL
LIN {X 0,Y 178.692,Z 418.225,A -85,B 0,C 180,E1 -22693.649,E2 -22693.649} C_VEL
LIN {X 0,Y 178.674,Z 418.221,A -85,B 0,C 180,E1 -22698.341,E2 -22698.341} C_VEL
LIN {X 0,Y 178.571,Z 418.26,A -85,B 0,C 180,E1 -22702.565,E2 -22702.565} C_VEL
LIN {X 0,Y 179.001,Z 420.996,A -85,B 0,C 180,E1 -22708.109,E2 -22708.109} C_VEL
LIN {X 0,Y 179.436,Z 423.921,A -85,B 0,C 180,E1 -22713.253,E2 -22713.253} C_VEL
LIN {X 0,Y 180.031,Z 427.353,A -85,B 0,C 180,E1 -22718.669,E2 -22718.669} C_VEL
LIN {X 0,Y 180.589,Z 429.848,A -85,B 0,C 180,E1 -22722.317,E2 -22722.317} C_VEL
LIN {X 0,Y 181.228,Z 433.199,A -85,B 0,C 180,E1 -22726.811,E2 -22726.811} C_VEL
LIN {X 0,Y 182.27,Z 436.292,A -85,B 0,C 180,E1 -22727.338,E2 -22727.338} C_VEL
LIN {X 0,Y 183.945,Z 439.06,A -85,B 0,C 180,E1 -22728.028,E2 -22728.028} C_VEL
LIN {X 0,Y 187.148,Z 446.802,A -85,B 0,C 180,E1 -22729.609,E2 -22729.609} C_VEL
LIN {X 0,Y 189.274,Z 456.028,A -85,B 0,C 180,E1 -22731.239,E2 -22731.239} C_VEL
LIN {X 0,Y 190.683,Z 465.776,A -85,B 0,C 180,E1 -22733.008,E2 -22733.008} C_VEL
LIN {X 0,Y 191.402,Z 476.785,A -85,B 0,C 180,E1 -22735.161,E2 -22735.161} C_VEL
LIN {X 0,Y 191.324,Z 487.035,A -85,B 0,C 180,E1 -22737.407,E2 -22737.407} C_VEL
LIN {X 0,Y 190.484,Z 496.751,A -85,B 0,C 180,E1 -22739.821,E2 -22739.821} C_VEL
LIN {X 0,Y 189.142,Z 503.58,A -85,B 0,C 180,E1 -22741.721,E2 -22741.721} C_VEL
LIN {X 0,Y 185.509,Z 513.271,A -85,B 0,C 180,E1 -22744.773,E2 -22744.773} C_VEL
LIN {X 0,Y 182.754,Z 521.016,A -85,B 0,C 180,E1 -22747.979,E2 -22747.979} C_VEL
LIN {X 0,Y 180.62,Z 526.319,A -85,B 0,C 180,E1 -22750.686,E2 -22750.686} C_VEL
LIN {X 0,Y 178.624,Z 531.469,A -85,B 0,C 180,E1 -22754.013,E2 -22754.013} C_VEL
LIN {X 0,Y 177.332,Z 535.489,A -85,B 0,C 180,E1 -22757.41,E2 -22757.41} C_VEL
LIN {X 0,Y 176.557,Z 538.471,A -85,B 0,C 180,E1 -22760.838,E2 -22760.838} C_VEL
LIN {X 0,Y 176.335,Z 539.898,A -85,B 0,C 180,E1 -22763.133,E2 -22763.133} C_VEL
LIN {X 0,Y 176.262,Z 540.922,A -85,B 0,C 180,E1 -22765.426,E2 -22765.426} C_VEL
LIN {X 0,Y 176.319,Z 541.552,A -85,B 0,C 180,E1 -22767.715,E2 -22767.715} C_VEL
LIN {X 0,Y 176.475,Z 541.779,A -85,B 0,C 180,E1 -22770,E2 -22770} C_VEL
LIN {X 0,Y 176.322,Z 541.541,A -85,B 0,C 180,E1 -22772.284,E2 -22772.284} C_VEL
LIN {X 0,Y 176.262,Z 540.906,A -85,B 0,C 180,E1 -22774.574,E2 -22774.574} C_VEL
LIN {X 0,Y 176.306,Z 539.874,A -85,B 0,C 180,E1 -22776.868,E2 -22776.868} C_VEL
LIN {X 0,Y 176.555,Z 538.437,A -85,B 0,C 180,E1 -22779.162,E2 -22779.162} C_VEL
LIN {X 0,Y 176.906,Z 536.921,A -85,B 0,C 180,E1 -22780.984,E2 -22780.984} C_VEL
LIN {X 0,Y 176.749,Z 535.247,A -85,B 0,C 180,E1 -22782.82,E2 -22782.82} C_VEL
LIN {X 0,Y 175.004,Z 531.939,A -85,B 0,C 180,E1 -22785.817,E2 -22785.817} C_VEL
LIN {X 0,Y 173.664,Z 527.911,A -85,B 0,C 180,E1 -22788.771,E2 -22788.771} C_VEL
LIN {X 0,Y 174.138,Z 525.105,A -85,B 0,C 180,E1 -22790.482,E2 -22790.482} C_VEL
LIN {X 0,Y 176.524,Z 519.29,A -85,B 0,C 180,E1 -22793.461,E2 -22793.461} C_VEL
LIN {X 0,Y 179.664,Z 511.196,A -85,B 0,C 180,E1 -22796.734,E2 -22796.734} C_VEL
LIN {X 0,Y 182.85,Z 502.968,A -85,B 0,C 180,E1 -22799.344,E2 -22799.344} C_VEL
LIN {X 0,Y 184.315,Z 493.897,A -85,B 0,C 180,E1 -22801.942,E2 -22801.942} C_VEL
LIN {X 0,Y 185.061,Z 483.829,A -85,B 0,C 180,E1 -22804.458,E2 -22804.458} C_VEL
LIN {X 0,Y 185.016,Z 473.423,A -85,B 0,C 180,E1 -22806.761,E2 -22806.761} C_VEL
LIN {X 0,Y 184.112,Z 462.692,A -85,B 0,C 180,E1 -22808.919,E2 -22808.919} C_VEL
LIN {X 0,Y 182.004,Z 451.026,A -85,B 0,C 180,E1 -22811.149,E2 -22811.149} C_VEL
LIN {X 0,Y 179.858,Z 445.277,A -85,B 0,C 180,E1 -22812.42,E2 -22812.42} C_VEL
LIN {X 0,Y 178.476,Z 442.23,A -85,B 0,C 180,E1 -22813.132,E2 -22813.132} C_VEL
LIN {X 0,Y 176.615,Z 438.216,A -85,B 0,C 180,E1 -22814.079,E2 -22814.079} C_VEL
LIN {X 0,Y 174.454,Z 434.649,A -85,B 0,C 180,E1 -22815.069,E2 -22815.069} C_VEL
LIN {X 0,Y 173.855,Z 432.5,A -85,B 0,C 180,E1 -22815.484,E2 -22815.484} C_VEL
LIN {X 0,Y 173.119,Z 429.114,A -85,B 0,C 180,E1 -22820.474,E2 -22820.474} C_VEL
LIN {X 0,Y 172.644,Z 426.161,A -85,B 0,C 180,E1 -22825.256,E2 -22825.256} C_VEL
LIN {X 0,Y 172.14,Z 423.135,A -85,B 0,C 180,E1 -22830.664,E2 -22830.664} C_VEL
LIN {X 0,Y 171.746,Z 420.553,A -85,B 0,C 180,E1 -22835.845,E2 -22835.845} C_VEL
LIN {X 0,Y 171.512,Z 419.12,A -85,B 0,C 180,E1 -22839.54,E2 -22839.54} C_VEL
LIN {X 0,Y 171.587,Z 419.112,A -85,B 0,C 180,E1 -22843.339,E2 -22843.339} C_VEL
LIN {X 0,Y 171.852,Z 419.08,A -85,B 0,C 180,E1 -22848.962,E2 -22848.962} C_VEL
LIN {X 0,Y 171.902,Z 419.075,A -85,B 0,C 180,E1 -22852.955,E2 -22852.955} C_VEL
LIN {X 0,Y 172.104,Z 419.048,A -85,B 0,C 180,E1 -22857.66,E2 -22857.66} C_VEL
LIN {X 0,Y 172.337,Z 419.018,A -85,B 0,C 180,E1 -22860,E2 -22860} C_VEL
LIN {X 0,Y 171.828,Z 419.08,A -85,B 0,C 180,E1 -22864.692,E2 -22864.692} C_VEL
LIN {X 0,Y 171.912,Z 419.07,A -85,B 0,C 180,E1 -22869.412,E2 -22869.412} C_VEL
LIN {X 0,Y 171.612,Z 419.109,A -85,B 0,C 180,E1 -22874.224,E2 -22874.224} C_VEL
LIN {X 0,Y 171.544,Z 419.115,A -85,B 0,C 180,E1 -22879.56,E2 -22879.56} C_VEL
LIN {X 0,Y 171.46,Z 419.128,A -85,B 0,C 180,E1 -22885.609,E2 -22885.609} C_VEL
LIN {X 0,Y 171.441,Z 419.13,A -85,B 0,C 180,E1 -22890.586,E2 -22890.586} C_VEL
LIN {X 0,Y 171.4,Z 419.135,A -85,B 0,C 180,E1 -22895.033,E2 -22895.033} C_VEL
LIN {X 0,Y 171.378,Z 419.138,A -85,B 0,C 180,E1 -22898.816,E2 -22898.816} C_VEL
LIN {X 0,Y 171.384,Z 419.264,A -85,B 0,C 180,E1 -22903.885,E2 -22903.885} C_VEL
LIN {X 0,Y 172.408,Z 421.994,A -85,B 0,C 180,E1 -22904.497,E2 -22904.497} C_VEL
LIN {X 0,Y 174.486,Z 424.45,A -85,B 0,C 180,E1 -22905.428,E2 -22905.428} C_VEL
LIN {X 0,Y 176.435,Z 427.742,A -85,B 0,C 180,E1 -22906.425,E2 -22906.425} C_VEL
LIN {X 0,Y 180.39,Z 434.998,A -85,B 0,C 180,E1 -22908.523,E2 -22908.523} C_VEL
LIN {X 0,Y 184.57,Z 445.427,A -85,B 0,C 180,E1 -22911.283,E2 -22911.283} C_VEL
LIN {X 0,Y 186.937,Z 453.975,A -85,B 0,C 180,E1 -22913.474,E2 -22913.474} C_VEL
LIN {X 0,Y 188.663,Z 463.721,A -85,B 0,C 180,E1 -22916.029,E2 -22916.029} C_VEL
LIN {X 0,Y 189.312,Z 471.029,A -85,B 0,C 180,E1 -22918.063,E2 -22918.063} C_VEL
LIN {X 0,Y 186.815,Z 479.564,A -85,B 0,C 180,E1 -22920.121,E2 -22920.121} C_VEL
LIN {X 0,Y 183.674,Z 488.289,A -85,B 0,C 180,E1 -22922.667,E2 -22922.667} C_VEL
LIN {X 0,Y 180.12,Z 496.864,A -85,B 0,C 180,E1 -22925.815,E2 -22925.815} C_VEL
LIN {X 0,Y 177.204,Z 503.685,A -85,B 0,C 180,E1 -22929.087,E2 -22929.087} C_VEL
LIN {X 0,Y 174.682,Z 509.147,A -85,B 0,C 180,E1 -22932.438,E2 -22932.438} C_VEL
LIN {X 0,Y 172.7,Z 513.427,A -85,B 0,C 180,E1 -22935.867,E2 -22935.867} C_VEL
LIN {X 0,Y 171.699,Z 515.687,A -85,B 0,C 180,E1 -22938.191,E2 -22938.191} C_VEL
LIN {X 0,Y 170.889,Z 517.668,A -85,B 0,C 180,E1 -22940.763,E2 -22940.763} C_VEL
LIN {X 0,Y 169.935,Z 519.875,A -85,B 0,C 180,E1 -22945.256,E2 -22945.256} C_VEL
LIN {X 0,Y 169.528,Z 520.707,A -85,B 0,C 180,E1 -22950,E2 -22950} C_VEL
LIN {X 0,Y 169.927,Z 519.925,A -85,B 0,C 180,E1 -22954.745,E2 -22954.745} C_VEL
LIN {X 0,Y 170.88,Z 517.622,A -85,B 0,C 180,E1 -22959.469,E2 -22959.469} C_VEL
LIN {X 0,Y 172.107,Z 514.778,A -85,B 0,C 180,E1 -22962.979,E2 -22962.979} C_VEL
LIN {X 0,Y 173.909,Z 510.91,A -85,B 0,C 180,E1 -22966.433,E2 -22966.433} C_VEL
LIN {X 0,Y 176.238,Z 505.914,A -85,B 0,C 180,E1 -22969.814,E2 -22969.814} C_VEL
LIN {X 0,Y 179.026,Z 499.617,A -85,B 0,C 180,E1 -22973.115,E2 -22973.115} C_VEL
LIN {X 0,Y 182.427,Z 491.725,A -85,B 0,C 180,E1 -22976.298,E2 -22976.298} C_VEL
LIN {X 0,Y 185.529,Z 483.681,A -85,B 0,C 180,E1 -22978.881,E2 -22978.881} C_VEL
LIN {X 0,Y 188.704,Z 473.874,A -85,B 0,C 180,E1 -22981.427,E2 -22981.427} C_VEL
LIN {X 0,Y 189.401,Z 471.609,A -85,B 0,C 180,E1 -22981.923,E2 -22981.923} C_VEL
LIN {X 0,Y 188.564,Z 462.342,A -85,B 0,C 180,E1 -22984.479,E2 -22984.479} C_VEL
LIN {X 0,Y 186.661,Z 452.537,A -85,B 0,C 180,E1 -22987.044,E2 -22987.044} C_VEL
LIN {X 0,Y 184.083,Z 443.895,A -85,B 0,C 180,E1 -22989.277,E2 -22989.277} C_VEL
LIN {X 0,Y 180.359,Z 435.037,A -85,B 0,C 180,E1 -22991.665,E2 -22991.665} C_VEL
LIN {X 0,Y 176.402,Z 427.804,A -85,B 0,C 180,E1 -22993.77,E2 -22993.77} C_VEL
LIN {X 0,Y 174.442,Z 424.56,A -85,B 0,C 180,E1 -22994.77,E2 -22994.77} C_VEL
LIN {X 0,Y 171.886,Z 421.13,A -85,B 0,C 180,E1 -22995.965,E2 -22995.965} C_VEL
LIN {X 0,Y 171.315,Z 419.145,A -85,B 0,C 180,E1 -22996.408,E2 -22996.408} C_VEL
LIN {X 0,Y 171.416,Z 419.13,A -85,B 0,C 180,E1 -23002.048,E2 -23002.048} C_VEL
LIN {X 0,Y 171.412,Z 419.126,A -85,B 0,C 180,E1 -23005.087,E2 -23005.087} C_VEL
LIN {X 0,Y 171.45,Z 419.128,A -85,B 0,C 180,E1 -23010.534,E2 -23010.534} C_VEL
LIN {X 0,Y 171.448,Z 419.127,A -85,B 0,C 180,E1 -23015.8,E2 -23015.8} C_VEL
LIN {X 0,Y 171.582,Z 419.11,A -85,B 0,C 180,E1 -23020.872,E2 -23020.872} C_VEL
LIN {X 0,Y 171.601,Z 419.109,A -85,B 0,C 180,E1 -23025.775,E2 -23025.775} C_VEL
LIN {X 0,Y 171.85,Z 419.08,A -85,B 0,C 180,E1 -23030.585,E2 -23030.585} C_VEL
LIN {X 0,Y 171.818,Z 419.083,A -85,B 0,C 180,E1 -23035.307,E2 -23035.307} C_VEL
LIN {X 0,Y 172.336,Z 419.023,A -85,B 0,C 180,E1 -23040,E2 -23040} C_VEL
LIN {X 0,Y 171.83,Z 419.085,A -85,B 0,C 180,E1 -23044.692,E2 -23044.692} C_VEL
LIN {X 0,Y 171.914,Z 419.071,A -85,B 0,C 180,E1 -23049.411,E2 -23049.411} C_VEL
LIN {X 0,Y 171.617,Z 419.106,A -85,B 0,C 180,E1 -23054.224,E2 -23054.224} C_VEL
LIN {X 0,Y 171.561,Z 419.115,A -85,B 0,C 180,E1 -23059.574,E2 -23059.574} C_VEL
LIN {X 0,Y 171.532,Z 419.245,A -85,B 0,C 180,E1 -23061.05,E2 -23061.05} C_VEL
LIN {X 0,Y 171.878,Z 421.45,A -85,B 0,C 180,E1 -23065.897,E2 -23065.897} C_VEL
LIN {X 0,Y 172.283,Z 424.117,A -85,B 0,C 180,E1 -23071.055,E2 -23071.055} C_VEL
LIN {X 0,Y 172.692,Z 426.695,A -85,B 0,C 180,E1 -23075.517,E2 -23075.517} C_VEL
LIN {X 0,Y 173.299,Z 429.816,A -85,B 0,C 180,E1 -23080.456,E2 -23080.456} C_VEL
LIN {X 0,Y 173.9,Z 432.629,A -85,B 0,C 180,E1 -23084.502,E2 -23084.502} C_VEL
LIN {X 0,Y 174.938,Z 435.634,A -85,B 0,C 180,E1 -23085.078,E2 -23085.078} C_VEL
LIN {X 0,Y 176.728,Z 438.479,A -85,B 0,C 180,E1 -23085.887,E2 -23085.887} C_VEL
LIN {X 0,Y 178.61,Z 442.473,A -85,B 0,C 180,E1 -23086.844,E2 -23086.844} C_VEL
LIN {X 0,Y 181.37,Z 449.06,A -85,B 0,C 180,E1 -23088.363,E2 -23088.363} C_VEL
LIN {X 0,Y 183.043,Z 455.855,A -85,B 0,C 180,E1 -23089.697,E2 -23089.697} C_VEL
LIN {X 0,Y 184.573,Z 466.567,A -85,B 0,C 180,E1 -23091.78,E2 -23091.78} C_VEL
LIN {X 0,Y 185.181,Z 478.089,A -85,B 0,C 180,E1 -23094.179,E2 -23094.179} C_VEL
LIN {X 0,Y 184.855,Z 489.08,A -85,B 0,C 180,E1 -23096.764,E2 -23096.764} C_VEL
LIN {X 0,Y 183.974,Z 497.36,A -85,B 0,C 180,E1 -23098.954,E2 -23098.954} C_VEL
LIN {X 0,Y 182.84,Z 503.144,A -85,B 0,C 180,E1 -23100.653,E2 -23100.653} C_VEL
LIN {X 0,Y 179.079,Z 512.839,A -85,B 0,C 180,E1 -23103.799,E2 -23103.799} C_VEL
LIN {X 0,Y 176.091,Z 520.579,A -85,B 0,C 180,E1 -23107.099,E2 -23107.099} C_VEL
LIN {X 0,Y 173.174,Z 527.725,A -85,B 0,C 180,E1 -23111.054,E2 -23111.054} C_VEL
LIN {X 0,Y 171.216,Z 532.485,A -85,B 0,C 180,E1 -23114.525,E2 -23114.525} C_VEL
LIN {X 0,Y 170.04,Z 536.145,A -85,B 0,C 180,E1 -23118.073,E2 -23118.073} C_VEL
LIN {X 0,Y 169.518,Z 538.037,A -85,B 0,C 180,E1 -23120.454,E2 -23120.454} C_VEL
LIN {X 0,Y 169.262,Z 539.465,A -85,B 0,C 180,E1 -23122.844,E2 -23122.844} C_VEL
LIN {X 0,Y 169.174,Z 540.613,A -85,B 0,C 180,E1 -23125.587,E2 -23125.587} C_VEL
LIN {X 0,Y 169.41,Z 541.349,A -85,B 0,C 180,E1 -23130,E2 -23130} C_VEL
LIN {X 0,Y 169.165,Z 540.608,A -85,B 0,C 180,E1 -23134.375,E2 -23134.375} C_VEL
LIN {X 0,Y 169.242,Z 539.44,A -85,B 0,C 180,E1 -23137.156,E2 -23137.156} C_VEL
LIN {X 0,Y 169.835,Z 536.718,A -85,B 0,C 180,E1 -23141.152,E2 -23141.152} C_VEL
LIN {X 0,Y 170.735,Z 533.752,A -85,B 0,C 180,E1 -23144.299,E2 -23144.299} C_VEL
LIN {X 0,Y 172.446,Z 529.353,A -85,B 0,C 180,E1 -23147.798,E2 -23147.798} C_VEL
LIN {X 0,Y 174.138,Z 525.105,A -85,B 0,C 180,E1 -23150.482,E2 -23150.482} C_VEL
LIN {X 0,Y 174.72,Z 522.133,A -85,B 0,C 180,E1 -23152.147,E2 -23152.147} C_VEL
LIN {X 0,Y 174.101,Z 516.918,A -85,B 0,C 180,E1 -23154.921,E2 -23154.921} C_VEL
LIN {X 0,Y 173.775,Z 511.153,A -85,B 0,C 180,E1 -23157.577,E2 -23157.577} C_VEL
LIN {X 0,Y 174.772,Z 507.281,A -85,B 0,C 180,E1 -23159.004,E2 -23159.004} C_VEL
LIN {X 0,Y 176.555,Z 502.523,A -85,B 0,C 180,E1 -23160.499,E2 -23160.499} C_VEL
LIN {X 0,Y 178.019,Z 493.438,A -85,B 0,C 180,E1 -23163.214,E2 -23163.214} C_VEL
LIN {X 0,Y 178.812,Z 483.528,A -85,B 0,C 180,E1 -23165.799,E2 -23165.799} C_VEL
LIN {X 0,Y 178.801,Z 473.343,A -85,B 0,C 180,E1 -23168.175,E2 -23168.175} C_VEL
LIN {X 0,Y 178.05,Z 463.275,A -85,B 0,C 180,E1 -23170.318,E2 -23170.318} C_VEL
LIN {X 0,Y 176.585,Z 454.342,A -85,B 0,C 180,E1 -23172.162,E2 -23172.162} C_VEL
LIN {X 0,Y 174.016,Z 447.245,A -85,B 0,C 180,E1 -23173.891,E2 -23173.891} C_VEL
LIN {X 0,Y 171.112,Z 441.4,A -85,B 0,C 180,E1 -23175.509,E2 -23175.509} C_VEL
LIN {X 0,Y 168.962,Z 437.07,A -85,B 0,C 180,E1 -23176.692,E2 -23176.692} C_VEL
LIN {X 0,Y 166.87,Z 433.534,A -85,B 0,C 180,E1 -23177.783,E2 -23177.783} C_VEL
LIN {X 0,Y 166.415,Z 431.882,A -85,B 0,C 180,E1 -23178.087,E2 -23178.087} C_VEL
LIN {X 0,Y 165.777,Z 428.469,A -85,B 0,C 180,E1 -23183.658,E2 -23183.658} C_VEL
LIN {X 0,Y 165.293,Z 425.318,A -85,B 0,C 180,E1 -23189.322,E2 -23189.322} C_VEL
LIN {X 0,Y 164.884,Z 422.632,A -85,B 0,C 180,E1 -23194.771,E2 -23194.771} C_VEL
LIN {X 0,Y 164.559,Z 420.402,A -85,B 0,C 180,E1 -23200.022,E2 -23200.022} C_VEL
LIN {X 0,Y 164.508,Z 419.993,A -85,B 0,C 180,E1 -23202.6,E2 -23202.6} C_VEL
LIN {X 0,Y 164.781,Z 419.961,A -85,B 0,C 180,E1 -23208.802,E2 -23208.802} C_VEL
LIN {X 0,Y 164.864,Z 419.952,A -85,B 0,C 180,E1 -23212.653,E2 -23212.653} C_VEL
LIN {X 0,Y 165.3,Z 419.894,A -85,B 0,C 180,E1 -23220,E2 -23220} C_VEL
LIN {X 0,Y 164.864,Z 419.946,A -85,B 0,C 180,E1 -23227.348,E2 -23227.348} C_VEL
LIN {X 0,Y 164.782,Z 419.959,A -85,B 0,C 180,E1 -23231.198,E2 -23231.198} C_VEL
LIN {X 0,Y 164.508,Z 419.994,A -85,B 0,C 180,E1 -23237.401,E2 -23237.401} C_VEL
LIN {X 0,Y 164.474,Z 419.998,A -85,B 0,C 180,E1 -23239.989,E2 -23239.989} C_VEL
LIN {X 0,Y 164.387,Z 420.008,A -85,B 0,C 180,E1 -23246.128,E2 -23246.128} C_VEL
LIN {X 0,Y 164.375,Z 420.008,A -85,B 0,C 180,E1 -23251.227,E2 -23251.227} C_VEL
LIN {X 0,Y 164.307,Z 420.011,A -85,B 0,C 180,E1 -23256.787,E2 -23256.787} C_VEL
LIN {X 0,Y 164.315,Z 420.061,A -85,B 0,C 180,E1 -23261.271,E2 -23261.271} C_VEL
LIN {X 0,Y 165.168,Z 422.627,A -85,B 0,C 180,E1 -23261.876,E2 -23261.876} C_VEL
LIN {X 0,Y 167.525,Z 425.454,A -85,B 0,C 180,E1 -23263.076,E2 -23263.076} C_VEL
LIN {X 0,Y 169.42,Z 428.642,A -85,B 0,C 180,E1 -23264.156,E2 -23264.156} C_VEL
LIN {X 0,Y 170.675,Z 430.517,A -85,B 0,C 180,E1 -23264.828,E2 -23264.828} C_VEL
LIN {X 0,Y 173.873,Z 436.113,A -85,B 0,C 180,E1 -23266.683,E2 -23266.683} C_VEL
LIN {X 0,Y 177.168,Z 443.596,A -85,B 0,C 180,E1 -23268.913,E2 -23268.913} C_VEL
LIN {X 0,Y 179.973,Z 452.29,A -85,B 0,C 180,E1 -23271.353,E2 -23271.353} C_VEL
LIN {X 0,Y 181.829,Z 461.046,A -85,B 0,C 180,E1 -23273.78,E2 -23273.78} C_VEL
LIN {X 0,Y 182.797,Z 469.712,A -85,B 0,C 180,E1 -23276.261,E2 -23276.261} C_VEL
LIN {X 0,Y 182.974,Z 472.746,A -85,B 0,C 180,E1 -23277.179,E2 -23277.179} C_VEL
LIN {X 0,Y 180.074,Z 481.869,A -85,B 0,C 180,E1 -23279.511,E2 -23279.511} C_VEL
LIN {X 0,Y 176.778,Z 490.308,A -85,B 0,C 180,E1 -23282.152,E2 -23282.152} C_VEL
LIN {X 0,Y 173.126,Z 498.517,A -85,B 0,C 180,E1 -23285.412,E2 -23285.412} C_VEL
LIN {X 0,Y 170.606,Z 504.118,A -85,B 0,C 180,E1 -23288.238,E2 -23288.238} C_VEL
LIN {X 0,Y 167.947,Z 509.58,A -85,B 0,C 180,E1 -23291.709,E2 -23291.709} C_VEL
LIN {X 0,Y 165.847,Z 513.859,A -85,B 0,C 180,E1 -23295.271,E2 -23295.271} C_VEL
LIN {X 0,Y 164.767,Z 516.12,A -85,B 0,C 180,E1 -23297.686,E2 -23297.686} C_VEL
LIN {X 0,Y 163.832,Z 518.252,A -85,B 0,C 180,E1 -23300.628,E2 -23300.628} C_VEL
LIN {X 0,Y 162.875,Z 520.307,A -85,B 0,C 180,E1 -23305.049,E2 -23305.049} C_VEL
LIN {X 0,Y 162.466,Z 521.137,A -85,B 0,C 180,E1 -23310,E2 -23310} C_VEL
LIN {X 0,Y 162.567,Z 520.941,A -85,B 0,C 180,E1 -23312.478,E2 -23312.478} C_VEL
LIN {X 0,Y 162.867,Z 520.356,A -85,B 0,C 180,E1 -23314.951,E2 -23314.951} C_VEL
LIN {X 0,Y 163.908,Z 518.052,A -85,B 0,C 180,E1 -23319.876,E2 -23319.876} C_VEL
LIN {X 0,Y 165.222,Z 515.208,A -85,B 0,C 180,E1 -23323.53,E2 -23323.53} C_VEL
LIN {X 0,Y 167.13,Z 511.34,A -85,B 0,C 180,E1 -23327.119,E2 -23327.119} C_VEL
LIN {X 0,Y 169.601,Z 506.343,A -85,B 0,C 180,E1 -23330.624,E2 -23330.624} C_VEL
LIN {X 0,Y 172.52,Z 500.047,A -85,B 0,C 180,E1 -23334.04,E2 -23334.04} C_VEL
LIN {X 0,Y 176.1,Z 492.154,A -85,B 0,C 180,E1 -23337.32,E2 -23337.32} C_VEL
LIN {X 0,Y 179.362,Z 484.109,A -85,B 0,C 180,E1 -23339.973,E2 -23339.973} C_VEL
LIN {X 0,Y 182.691,Z 474.302,A -85,B 0,C 180,E1 -23342.587,E2 -23342.587} C_VEL
LIN {X 0,Y 183.02,Z 472.232,A -85,B 0,C 180,E1 -23343.128,E2 -23343.128} C_VEL
LIN {X 0,Y 182.401,Z 464.23,A -85,B 0,C 180,E1 -23345.469,E2 -23345.469} C_VEL
LIN {X 0,Y 180.74,Z 455.01,A -85,B 0,C 180,E1 -23348.057,E2 -23348.057} C_VEL
LIN {X 0,Y 178.37,Z 446.797,A -85,B 0,C 180,E1 -23350.35,E2 -23350.35} C_VEL
LIN {X 0,Y 175.594,Z 439.771,A -85,B 0,C 180,E1 -23352.4,E2 -23352.4} C_VEL
LIN {X 0,Y 171.675,Z 432.411,A -85,B 0,C 180,E1 -23354.763,E2 -23354.763} C_VEL
LIN {X 0,Y 169.51,Z 428.831,A -85,B 0,C 180,E1 -23355.992,E2 -23355.992} C_VEL
LIN {X 0,Y 167.533,Z 425.568,A -85,B 0,C 180,E1 -23357.115,E2 -23357.115} C_VEL
LIN {X 0,Y 166.405,Z 424.209,A -85,B 0,C 180,E1 -23357.692,E2 -23357.692} C_VEL
LIN {X 0,Y 164.844,Z 421.971,A -85,B 0,C 180,E1 -23358.535,E2 -23358.535} C_VEL
LIN {X 0,Y 164.327,Z 420.014,A -85,B 0,C 180,E1 -23358.987,E2 -23358.987} C_VEL
LIN {X 0,Y 164.345,Z 420.006,A -85,B 0,C 180,E1 -23364.343,E2 -23364.343} C_VEL
LIN {X 0,Y 164.392,Z 420.008,A -85,B 0,C 180,E1 -23369.135,E2 -23369.135} C_VEL
LIN {X 0,Y 164.409,Z 420.003,A -85,B 0,C 180,E1 -23374.693,E2 -23374.693} C_VEL
LIN {X 0,Y 164.487,Z 419.994,A -85,B 0,C 180,E1 -23380.051,E2 -23380.051} C_VEL
LIN {X 0,Y 164.549,Z 419.989,A -85,B 0,C 180,E1 -23385.151,E2 -23385.151} C_VEL
LIN {X 0,Y 164.771,Z 419.96,A -85,B 0,C 180,E1 -23390.176,E2 -23390.176} C_VEL
LIN {X 0,Y 164.833,Z 419.952,A -85,B 0,C 180,E1 -23392.651,E2 -23392.651} C_VEL
LIN {X 0,Y 165.051,Z 419.929,A -85,B 0,C 180,E1 -23397.559,E2 -23397.559} C_VEL
LIN {X 0,Y 165.299,Z 419.9,A -85,B 0,C 180,E1 -23400,E2 -23400} C_VEL
LIN {X 0,Y 164.78,Z 419.964,A -85,B 0,C 180,E1 -23404.893,E2 -23404.893} C_VEL
LIN {X 0,Y 164.866,Z 419.951,A -85,B 0,C 180,E1 -23407.347,E2 -23407.347} C_VEL
LIN {X 0,Y 164.783,Z 419.959,A -85,B 0,C 180,E1 -23411.198,E2 -23411.198} C_VEL
LIN {X 0,Y 164.522,Z 419.98,A -85,B 0,C 180,E1 -23417.399,E2 -23417.399} C_VEL
LIN {X 0,Y 164.584,Z 420.488,A -85,B 0,C 180,E1 -23420.041,E2 -23420.041} C_VEL
LIN {X 0,Y 164.886,Z 422.696,A -85,B 0,C 180,E1 -23425.229,E2 -23425.229} C_VEL
LIN {X 0,Y 165.294,Z 425.381,A -85,B 0,C 180,E1 -23430.678,E2 -23430.678} C_VEL
LIN {X 0,Y 165.782,Z 428.587,A -85,B 0,C 180,E1 -23436.406,E2 -23436.406} C_VEL
LIN {X 0,Y 166.468,Z 431.959,A -85,B 0,C 180,E1 -23441.832,E2 -23441.832} C_VEL
LIN {X 0,Y 167.505,Z 434.888,A -85,B 0,C 180,E1 -23442.472,E2 -23442.472} C_VEL
LIN {X 0,Y 169.744,Z 438.349,A -85,B 0,C 180,E1 -23443.597,E2 -23443.597} C_VEL
LIN {X 0,Y 171.732,Z 442.318,A -85,B 0,C 180,E1 -23444.699,E2 -23444.699} C_VEL
LIN {X 0,Y 175.62,Z 451.095,A -85,B 0,C 180,E1 -23446.997,E2 -23446.997} C_VEL
LIN {X 0,Y 177.205,Z 457.211,A -85,B 0,C 180,E1 -23448.355,E2 -23448.355} C_VEL
LIN {X 0,Y 178.623,Z 468.716,A -85,B 0,C 180,E1 -23450.762,E2 -23450.762} C_VEL
LIN {X 0,Y 178.965,Z 479.496,A -85,B 0,C 180,E1 -23453.177,E2 -23453.177} C_VEL
LIN {X 0,Y 178.456,Z 489.987,A -85,B 0,C 180,E1 -23455.795,E2 -23455.795} C_VEL
LIN {X 0,Y 177.309,Z 498.903,A -85,B 0,C 180,E1 -23458.318,E2 -23458.318} C_VEL
LIN {X 0,Y 175.993,Z 504.509,A -85,B 0,C 180,E1 -23460.055,E2 -23460.055} C_VEL
LIN {X 0,Y 172.108,Z 513.789,A -85,B 0,C 180,E1 -23463.308,E2 -23463.308} C_VEL
LIN {X 0,Y 169.093,Z 521.278,A -85,B 0,C 180,E1 -23466.743,E2 -23466.743} C_VEL
LIN {X 0,Y 166.405,Z 527.289,A -85,B 0,C 180,E1 -23470.252,E2 -23470.252} C_VEL
LIN {X 0,Y 164.359,Z 532.052,A -85,B 0,C 180,E1 -23473.862,E2 -23473.862} C_VEL
LIN {X 0,Y 163.07,Z 535.711,A -85,B 0,C 180,E1 -23477.555,E2 -23477.555} C_VEL
LIN {X 0,Y 162.479,Z 537.603,A -85,B 0,C 180,E1 -23480.036,E2 -23480.036} C_VEL
LIN {X 0,Y 162.187,Z 539.031,A -85,B 0,C 180,E1 -23482.53,E2 -23482.53} C_VEL
LIN {X 0,Y 162.098,Z 540.287,A -85,B 0,C 180,E1 -23485.71,E2 -23485.71} C_VEL
LIN {X 0,Y 162.323,Z 540.917,A -85,B 0,C 180,E1 -23490,E2 -23490} C_VEL
LIN {X 0,Y 162.082,Z 540.293,A -85,B 0,C 180,E1 -23494.213,E2 -23494.213} C_VEL
LIN {X 0,Y 162.174,Z 539.006,A -85,B 0,C 180,E1 -23497.47,E2 -23497.47} C_VEL
LIN {X 0,Y 162.478,Z 537.567,A -85,B 0,C 180,E1 -23499.963,E2 -23499.963} C_VEL
LIN {X 0,Y 163.396,Z 534.566,A -85,B 0,C 180,E1 -23503.684,E2 -23503.684} C_VEL
LIN {X 0,Y 164.973,Z 530.53,A -85,B 0,C 180,E1 -23507.35,E2 -23507.35} C_VEL
LIN {X 0,Y 167.632,Z 524.347,A -85,B 0,C 180,E1 -23511.521,E2 -23511.521} C_VEL
LIN {X 0,Y 170.167,Z 518.29,A -85,B 0,C 180,E1 -23514.686,E2 -23514.686} C_VEL
LIN {X 0,Y 173.312,Z 510.758,A -85,B 0,C 180,E1 -23517.797,E2 -23517.797} C_VEL
LIN {X 0,Y 174.772,Z 507.281,A -85,B 0,C 180,E1 -23519.004,E2 -23519.004} C_VEL
